LIN {X 0.170,Y -404.553,Z 1346.396,A 0.000,B 0.000,C 90.000,E1 287.221} C_DIS
LIN {X -0.116,Y -404.761,Z 1346.394,A 0.000,B 0.000,C 90.000,E1 286.913} C_DIS
LIN {X -0.219,Y -406.031,Z 1346.365,A 0.000,B 0.000,C 90.000,E1 281.715} C_DIS
LIN {X -0.210,Y -406.144,Z 1346.363,A 0.000,B 0.000,C 90.000,E1 281.366} C_DIS
LIN {X -0.106,Y -405.652,Z 1346.334,A 0.000,B 0.000,C 90.000,E1 276.144} C_DIS
LIN {X -0.101,Y -405.611,Z 1346.332,A 0.000,B 0.000,C 90.000,E1 275.796} C_DIS
LIN {X -0.028,Y -403.552,Z 1346.305,A 0.000,B 0.000,C 90.000,E1 270.917} C_DIS
LIN {X -0.092,Y -403.056,Z 1346.301,A 0.000,B 0.000,C 90.000,E1 270.229} C_DIS
LIN {X 0.132,Y -399.017,Z 1346.272,A 0.000,B 0.000,C 90.000,E1 264.951} C_DIS
LIN {X 0.026,Y -397.651,Z 1346.266,A 0.000,B 0.000,C 90.000,E1 263.913} C_DIS
LIN {X -0.094,Y -392.933,Z 1346.241,A 0.000,B 0.000,C 90.000,E1 259.342} C_DIS
LIN {X -0.136,Y -392.480,Z 1346.239,A 0.000,B 0.000,C 90.000,E1 258.993} C_DIS
LIN {X 0.013,Y -386.123,Z 1346.213,A 0.000,B 0.000,C 90.000,E1 254.338} C_DIS
LIN {X -0.028,Y -384.992,Z 1346.207,A 0.000,B 0.000,C 90.000,E1 253.268} C_DIS
LIN {X -0.154,Y -378.133,Z 1346.183,A 0.000,B 0.000,C 90.000,E1 248.954} C_DIS
LIN {X -0.065,Y -376.372,Z 1346.175,A 0.000,B 0.000,C 90.000,E1 247.486} C_DIS
LIN {X 0.060,Y -375.883,Z 1346.173,A 0.000,B 0.000,C 90.000,E1 247.102} C_DIS
LIN {X 0.010,Y -369.104,Z 1346.151,A 0.000,B 0.000,C 90.000,E1 243.076} C_DIS
LIN {X 0.089,Y -366.257,Z 1346.138,A 0.000,B 0.000,C 90.000,E1 240.845} C_DIS
LIN {X 0.050,Y -358.852,Z 1346.113,A 0.000,B 0.000,C 90.000,E1 236.373} C_DIS
LIN {X 0.038,Y -356.042,Z 1346.101,A 0.000,B 0.000,C 90.000,E1 234.116} C_DIS
LIN {X 0.034,Y -348.479,Z 1346.073,A 0.000,B 0.000,C 90.000,E1 229.175} C_DIS
LIN {X 0.095,Y -345.898,Z 1346.061,A 0.000,B 0.000,C 90.000,E1 226.863} C_DIS
LIN {X 0.062,Y -339.123,Z 1346.033,A 0.000,B 0.000,C 90.000,E1 221.838} C_DIS
LIN {X 0.145,Y -336.957,Z 1346.020,A 0.000,B 0.000,C 90.000,E1 219.483} C_DIS
LIN {X -0.034,Y -334.079,Z 1346.007,A 0.000,B 0.000,C 90.000,E1 217.202} C_DIS
LIN {X -0.051,Y -334.075,Z 1346.007,A 0.000,B 0.000,C 90.000,E1 217.202} C_DIS
LIN {X 0.031,Y -350.965,Z 1345.996,A 0.000,B 0.000,C 90.000,E1 215.185} C_DIS
LIN {X -0.024,Y -369.522,Z 1345.985,A 0.000,B 0.000,C 90.000,E1 213.245} C_DIS
LIN {X 0.079,Y -388.468,Z 1345.975,A 0.000,B 0.000,C 90.000,E1 211.465} C_DIS
LIN {X 0.012,Y -409.375,Z 1345.965,A 0.000,B 0.000,C 90.000,E1 209.745} C_DIS
LIN {X -0.255,Y -432.257,Z 1345.956,A 0.000,B 0.000,C 90.000,E1 208.103} C_DIS
LIN {X 0.054,Y -445.485,Z 1345.951,A 0.000,B 0.000,C 90.000,E1 207.180} C_DIS
LIN {X -0.207,Y -447.707,Z 1345.950,A 0.000,B 0.000,C 90.000,E1 207.001} C_DIS
LIN {X -0.015,Y -449.218,Z 1345.948,A 0.000,B 0.000,C 90.000,E1 206.693} C_DIS
LIN {X 0.051,Y -450.444,Z 1345.947,A 0.000,B 0.000,C 90.000,E1 206.360} C_DIS
LIN {X -0.075,Y -451.427,Z 1345.945,A 0.000,B 0.000,C 90.000,E1 206.052} C_DIS
LIN {X -0.118,Y -453.031,Z 1345.941,A 0.000,B 0.000,C 90.000,E1 205.412} C_DIS
LIN {X -0.151,Y -454.100,Z 1345.938,A 0.000,B 0.000,C 90.000,E1 204.771} C_DIS
LIN {X 0.033,Y -455.778,Z 1345.930,A 0.000,B 0.000,C 90.000,E1 203.462} C_DIS
LIN {X 0.063,Y -458.055,Z 1345.920,A 0.000,B 0.000,C 90.000,E1 201.535} C_DIS
LIN {X -0.205,Y -459.177,Z 1345.914,A 0.000,B 0.000,C 90.000,E1 200.610} C_DIS
LIN {X -0.077,Y -461.720,Z 1345.902,A 0.000,B 0.000,C 90.000,E1 198.362} C_DIS
LIN {X -0.023,Y -462.750,Z 1345.897,A 0.000,B 0.000,C 90.000,E1 197.402} C_DIS
LIN {X 0.202,Y -464.303,Z 1345.888,A 0.000,B 0.000,C 90.000,E1 195.788} C_DIS
LIN {X 0.054,Y -466.380,Z 1345.876,A 0.000,B 0.000,C 90.000,E1 193.592} C_DIS
LIN {X -0.076,Y -468.219,Z 1345.865,A 0.000,B 0.000,C 90.000,E1 191.715} C_DIS
LIN {X -0.254,Y -470.044,Z 1345.855,A 0.000,B 0.000,C 90.000,E1 189.849} C_DIS
LIN {X 0.135,Y -470.925,Z 1345.849,A 0.000,B 0.000,C 90.000,E1 188.859} C_DIS
LIN {X 0.107,Y -472.206,Z 1345.841,A 0.000,B 0.000,C 90.000,E1 187.296} C_DIS
LIN {X -0.248,Y -473.043,Z 1345.834,A 0.000,B 0.000,C 90.000,E1 186.087} C_DIS
LIN {X 0.107,Y -473.449,Z 1345.828,A 0.000,B 0.000,C 90.000,E1 185.106} C_DIS
LIN {X 0.241,Y -473.891,Z 1345.822,A 0.000,B 0.000,C 90.000,E1 183.841} C_DIS
LIN {X -0.126,Y -474.134,Z 1345.815,A 0.000,B 0.000,C 90.000,E1 182.636} C_DIS
LIN {X -0.016,Y -474.024,Z 1345.808,A 0.000,B 0.000,C 90.000,E1 181.375} C_DIS
LIN {X -0.181,Y -473.720,Z 1345.802,A 0.000,B 0.000,C 90.000,E1 180.458} C_DIS
LIN {X 0.126,Y -473.146,Z 1345.797,A 0.000,B 0.000,C 90.000,E1 179.484} C_DIS
LIN {X 0.206,Y -472.087,Z 1345.790,A 0.000,B 0.000,C 90.000,E1 178.224} C_DIS
LIN {X -0.192,Y -470.752,Z 1345.783,A 0.000,B 0.000,C 90.000,E1 177.020} C_DIS
LIN {X 0.091,Y -469.526,Z 1345.778,A 0.000,B 0.000,C 90.000,E1 176.045} C_DIS
LIN {X -0.071,Y -467.856,Z 1345.773,A 0.000,B 0.000,C 90.000,E1 175.122} C_DIS
LIN {X -0.043,Y -466.543,Z 1345.769,A 0.000,B 0.000,C 90.000,E1 174.489} C_DIS
LIN {X -0.026,Y -464.954,Z 1345.766,A 0.000,B 0.000,C 90.000,E1 173.856} C_DIS
LIN {X 0.182,Y -464.058,Z 1345.764,A 0.000,B 0.000,C 90.000,E1 173.514} C_DIS
LIN {X -0.036,Y -460.479,Z 1345.759,A 0.000,B 0.000,C 90.000,E1 172.591} C_DIS
LIN {X -0.010,Y -457.660,Z 1345.755,A 0.000,B 0.000,C 90.000,E1 171.951} C_DIS
LIN {X 0.143,Y -452.767,Z 1345.750,A 0.000,B 0.000,C 90.000,E1 170.971} C_DIS
LIN {X 0.244,Y -448.171,Z 1345.745,A 0.000,B 0.000,C 90.000,E1 170.151} C_DIS
LIN {X -0.083,Y -441.753,Z 1345.740,A 0.000,B 0.000,C 90.000,E1 169.218} C_DIS
LIN {X -0.218,Y -430.582,Z 1345.731,A 0.000,B 0.000,C 90.000,E1 167.589} C_DIS
LIN {X -0.058,Y -420.777,Z 1345.723,A 0.000,B 0.000,C 90.000,E1 166.061} C_DIS
LIN {X -0.011,Y -413.262,Z 1345.716,A 0.000,B 0.000,C 90.000,E1 164.866} C_DIS
LIN {X -0.056,Y -409.100,Z 1345.711,A 0.000,B 0.000,C 90.000,E1 164.031} C_DIS
LIN {X 0.156,Y -407.795,Z 1345.707,A 0.000,B 0.000,C 90.000,E1 163.268} C_DIS
LIN {X 0.118,Y -407.794,Z 1345.707,A 0.000,B 0.000,C 90.000,E1 163.268} C_DIS
LIN {X -0.092,Y -408.375,Z 1345.706,A 0.000,B 0.000,C 90.000,E1 163.087} C_DIS
LIN {X -0.078,Y -411.298,Z 1345.704,A 0.000,B 0.000,C 90.000,E1 162.653} C_DIS
LIN {X 0.071,Y -415.884,Z 1345.701,A 0.000,B 0.000,C 90.000,E1 162.127} C_DIS
LIN {X -0.127,Y -422.793,Z 1345.697,A 0.000,B 0.000,C 90.000,E1 161.511} C_DIS
LIN {X -0.205,Y -446.107,Z 1345.687,A 0.000,B 0.000,C 90.000,E1 159.699} C_DIS
LIN {X -0.083,Y -457.186,Z 1345.682,A 0.000,B 0.000,C 90.000,E1 158.847} C_DIS
LIN {X 0.010,Y -464.943,Z 1345.679,A 0.000,B 0.000,C 90.000,E1 158.230} C_DIS
LIN {X 0.070,Y -473.995,Z 1345.675,A 0.000,B 0.000,C 90.000,E1 157.486} C_DIS
LIN {X 0.028,Y -481.379,Z 1345.672,A 0.000,B 0.000,C 90.000,E1 156.869} C_DIS
LIN {X 0.099,Y -488.371,Z 1345.668,A 0.000,B 0.000,C 90.000,E1 156.230} C_DIS
LIN {X -0.060,Y -493.954,Z 1345.665,A 0.000,B 0.000,C 90.000,E1 155.717} C_DIS
LIN {X 0.040,Y -499.316,Z 1345.662,A 0.000,B 0.000,C 90.000,E1 155.177} C_DIS
LIN {X 0.115,Y -504.686,Z 1345.659,A 0.000,B 0.000,C 90.000,E1 154.613} C_DIS
LIN {X 0.140,Y -511.236,Z 1345.655,A 0.000,B 0.000,C 90.000,E1 153.896} C_DIS
LIN {X -0.009,Y -517.453,Z 1345.651,A 0.000,B 0.000,C 90.000,E1 153.179} C_DIS
LIN {X -0.220,Y -521.911,Z 1345.648,A 0.000,B 0.000,C 90.000,E1 152.615} C_DIS
LIN {X -0.159,Y -525.998,Z 1345.645,A 0.000,B 0.000,C 90.000,E1 152.025} C_DIS
LIN {X -0.067,Y -529.614,Z 1345.641,A 0.000,B 0.000,C 90.000,E1 151.435} C_DIS
LIN {X -0.093,Y -533.283,Z 1345.637,A 0.000,B 0.000,C 90.000,E1 150.717} C_DIS
LIN {X 0.056,Y -535.734,Z 1345.634,A 0.000,B 0.000,C 90.000,E1 150.127} C_DIS
LIN {X 0.220,Y -537.845,Z 1345.631,A 0.000,B 0.000,C 90.000,E1 149.537} C_DIS
LIN {X -0.343,Y -540.583,Z 1345.626,A 0.000,B 0.000,C 90.000,E1 148.742} C_DIS
LIN {X 0.135,Y -542.263,Z 1345.623,A 0.000,B 0.000,C 90.000,E1 148.122} C_DIS
LIN {X -0.095,Y -544.312,Z 1345.618,A 0.000,B 0.000,C 90.000,E1 147.296} C_DIS
LIN {X 0.155,Y -546.038,Z 1345.614,A 0.000,B 0.000,C 90.000,E1 146.421} C_DIS
LIN {X -0.035,Y -547.498,Z 1345.609,A 0.000,B 0.000,C 90.000,E1 145.595} C_DIS
LIN {X 0.054,Y -548.334,Z 1345.606,A 0.000,B 0.000,C 90.000,E1 145.022} C_DIS
LIN {X -0.062,Y -549.657,Z 1345.599,A 0.000,B 0.000,C 90.000,E1 143.909} C_DIS
LIN {X 0.162,Y -550.705,Z 1345.593,A 0.000,B 0.000,C 90.000,E1 142.763} C_DIS
LIN {X -0.035,Y -551.461,Z 1345.587,A 0.000,B 0.000,C 90.000,E1 141.662} C_DIS
LIN {X 0.379,Y -552.907,Z 1345.575,A 0.000,B 0.000,C 90.000,E1 139.380} C_DIS
LIN {X -0.141,Y -553.900,Z 1345.565,A 0.000,B 0.000,C 90.000,E1 137.757} C_DIS
LIN {X -0.205,Y -555.288,Z 1345.554,A 0.000,B 0.000,C 90.000,E1 135.810} C_DIS
LIN {X -0.220,Y -555.835,Z 1345.552,A 0.000,B 0.000,C 90.000,E1 135.324} C_DIS
LIN {X 0.002,Y -556.345,Z 1345.551,A 0.000,B 0.000,C 90.000,E1 135.162} C_DIS
LIN {X -0.102,Y -557.120,Z 1345.549,A 0.000,B 0.000,C 90.000,E1 134.838} C_DIS
LIN {X -0.144,Y -557.146,Z 1345.549,A 0.000,B 0.000,C 90.000,E1 134.838} C_DIS
LIN {X 0.106,Y -558.859,Z 1345.548,A 0.000,B 0.000,C 90.000,E1 134.595} C_DIS
LIN {X 0.291,Y -560.046,Z 1345.547,A 0.000,B 0.000,C 90.000,E1 134.514} C_DIS
LIN {X -0.276,Y -563.592,Z 1345.547,A 0.000,B 0.000,C 90.000,E1 134.433} C_DIS
LIN {X -0.342,Y -570.141,Z 1345.546,A 0.000,B 0.000,C 90.000,E1 134.271} C_DIS
LIN {X 0.031,Y -576.254,Z 1345.545,A 0.000,B 0.000,C 90.000,E1 134.028} C_DIS
LIN {X -0.356,Y -579.013,Z 1345.544,A 0.000,B 0.000,C 90.000,E1 133.947} C_DIS
LIN {X -0.199,Y -581.849,Z 1345.543,A 0.000,B 0.000,C 90.000,E1 133.785} C_DIS
LIN {X -0.033,Y -587.833,Z 1345.541,A 0.000,B 0.000,C 90.000,E1 133.419} C_DIS
LIN {X 0.071,Y -593.487,Z 1345.539,A 0.000,B 0.000,C 90.000,E1 133.014} C_DIS
LIN {X 0.242,Y -600.274,Z 1345.536,A 0.000,B 0.000,C 90.000,E1 132.447} C_DIS
LIN {X 0.007,Y -604.275,Z 1345.534,A 0.000,B 0.000,C 90.000,E1 132.123} C_DIS
LIN {X 0.042,Y -608.133,Z 1345.532,A 0.000,B 0.000,C 90.000,E1 131.757} C_DIS
LIN {X -0.044,Y -614.106,Z 1345.529,A 0.000,B 0.000,C 90.000,E1 131.148} C_DIS
LIN {X -0.248,Y -617.693,Z 1345.526,A 0.000,B 0.000,C 90.000,E1 130.782} C_DIS
LIN {X -0.047,Y -621.112,Z 1345.524,A 0.000,B 0.000,C 90.000,E1 130.378} C_DIS
LIN {X -0.085,Y -629.579,Z 1345.519,A 0.000,B 0.000,C 90.000,E1 129.358} C_DIS
LIN {X 0.281,Y -633.561,Z 1345.516,A 0.000,B 0.000,C 90.000,E1 128.830} C_DIS
LIN {X 0.010,Y -640.999,Z 1345.510,A 0.000,B 0.000,C 90.000,E1 127.855} C_DIS
LIN {X -0.169,Y -647.317,Z 1345.505,A 0.000,B 0.000,C 90.000,E1 126.996} C_DIS
LIN {X -0.109,Y -654.109,Z 1345.500,A 0.000,B 0.000,C 90.000,E1 126.011} C_DIS
LIN {X 0.081,Y -659.401,Z 1345.495,A 0.000,B 0.000,C 90.000,E1 125.152} C_DIS
LIN {X -0.317,Y -661.520,Z 1345.493,A 0.000,B 0.000,C 90.000,E1 124.818} C_DIS
LIN {X -0.274,Y -664.233,Z 1345.491,A 0.000,B 0.000,C 90.000,E1 124.326} C_DIS
LIN {X -0.152,Y -667.222,Z 1345.487,A 0.000,B 0.000,C 90.000,E1 123.706} C_DIS
LIN {X -0.078,Y -669.440,Z 1345.484,A 0.000,B 0.000,C 90.000,E1 123.214} C_DIS
LIN {X 0.158,Y -672.291,Z 1345.480,A 0.000,B 0.000,C 90.000,E1 122.467} C_DIS
LIN {X 0.067,Y -674.753,Z 1345.476,A 0.000,B 0.000,C 90.000,E1 121.750} C_DIS
LIN {X -0.042,Y -677.575,Z 1345.471,A 0.000,B 0.000,C 90.000,E1 120.797} C_DIS
LIN {X -0.069,Y -679.277,Z 1345.467,A 0.000,B 0.000,C 90.000,E1 120.079} C_DIS
LIN {X 0.259,Y -680.584,Z 1345.463,A 0.000,B 0.000,C 90.000,E1 119.333} C_DIS
LIN {X 0.061,Y -681.180,Z 1345.460,A 0.000,B 0.000,C 90.000,E1 118.871} C_DIS
LIN {X -0.134,Y -681.586,Z 1345.458,A 0.000,B 0.000,C 90.000,E1 118.409} C_DIS
LIN {X -0.125,Y -681.905,Z 1345.454,A 0.000,B 0.000,C 90.000,E1 117.692} C_DIS
LIN {X 0.183,Y -681.926,Z 1345.450,A 0.000,B 0.000,C 90.000,E1 116.950} C_DIS
LIN {X -0.208,Y -681.638,Z 1345.445,A 0.000,B 0.000,C 90.000,E1 116.027} C_DIS
LIN {X 0.113,Y -681.090,Z 1345.441,A 0.000,B 0.000,C 90.000,E1 115.283} C_DIS
LIN {X -0.097,Y -680.508,Z 1345.438,A 0.000,B 0.000,C 90.000,E1 114.823} C_DIS
LIN {X 0.022,Y -679.537,Z 1345.435,A 0.000,B 0.000,C 90.000,E1 114.335} C_DIS
LIN {X 0.415,Y -677.762,Z 1345.433,A 0.000,B 0.000,C 90.000,E1 113.823} C_DIS
LIN {X -0.286,Y -676.651,Z 1345.431,A 0.000,B 0.000,C 90.000,E1 113.643} C_DIS
LIN {X 0.184,Y -673.160,Z 1345.429,A 0.000,B 0.000,C 90.000,E1 113.153} C_DIS
LIN {X -0.346,Y -672.106,Z 1345.428,A 0.000,B 0.000,C 90.000,E1 113.078} C_DIS
LIN {X -0.258,Y -670.472,Z 1345.427,A 0.000,B 0.000,C 90.000,E1 112.950} C_DIS
LIN {X 0.297,Y -663.898,Z 1345.425,A 0.000,B 0.000,C 90.000,E1 112.514} C_DIS
LIN {X -0.134,Y -661.646,Z 1345.425,A 0.000,B 0.000,C 90.000,E1 112.461} C_DIS
LIN {X 0.299,Y -658.561,Z 1345.424,A 0.000,B 0.000,C 90.000,E1 112.333} C_DIS
LIN {X 0.252,Y -650.352,Z 1345.423,A 0.000,B 0.000,C 90.000,E1 112.153} C_DIS
LIN {X -0.169,Y -638.300,Z 1345.422,A 0.000,B 0.000,C 90.000,E1 111.950} C_DIS
LIN {X 0.373,Y -638.087,Z 1345.422,A 0.000,B 0.000,C 90.000,E1 111.897} C_DIS
LIN {X -0.028,Y -644.468,Z 1345.418,A 0.000,B 0.000,C 90.000,E1 111.153} C_DIS
LIN {X -0.166,Y -647.479,Z 1345.416,A 0.000,B 0.000,C 90.000,E1 110.791} C_DIS
LIN {X -0.291,Y -650.339,Z 1345.413,A 0.000,B 0.000,C 90.000,E1 110.429} C_DIS
LIN {X 0.343,Y -654.989,Z 1345.409,A 0.000,B 0.000,C 90.000,E1 109.631} C_DIS
LIN {X 0.261,Y -657.007,Z 1345.407,A 0.000,B 0.000,C 90.000,E1 109.268} C_DIS
LIN {X 0.074,Y -660.098,Z 1345.404,A 0.000,B 0.000,C 90.000,E1 108.671} C_DIS
LIN {X -0.034,Y -663.306,Z 1345.400,A 0.000,B 0.000,C 90.000,E1 107.946} C_DIS
LIN {X -0.115,Y -666.150,Z 1345.396,A 0.000,B 0.000,C 90.000,E1 107.221} C_DIS
LIN {X -0.092,Y -667.945,Z 1345.393,A 0.000,B 0.000,C 90.000,E1 106.732} C_DIS
LIN {X -0.325,Y -670.274,Z 1345.389,A 0.000,B 0.000,C 90.000,E1 106.024} C_DIS
LIN {X 0.297,Y -672.261,Z 1345.385,A 0.000,B 0.000,C 90.000,E1 105.245} C_DIS
LIN {X 0.171,Y -673.414,Z 1345.382,A 0.000,B 0.000,C 90.000,E1 104.773} C_DIS
LIN {X 0.055,Y -674.387,Z 1345.380,A 0.000,B 0.000,C 90.000,E1 104.300} C_DIS
LIN {X -0.056,Y -675.122,Z 1345.377,A 0.000,B 0.000,C 90.000,E1 103.828} C_DIS
LIN {X -0.213,Y -675.835,Z 1345.373,A 0.000,B 0.000,C 90.000,E1 103.119} C_DIS
LIN {X 0.344,Y -676.119,Z 1345.370,A 0.000,B 0.000,C 90.000,E1 102.591} C_DIS
LIN {X 0.190,Y -676.057,Z 1345.366,A 0.000,B 0.000,C 90.000,E1 101.883} C_DIS
LIN {X -0.049,Y -675.823,Z 1345.364,A 0.000,B 0.000,C 90.000,E1 101.422} C_DIS
LIN {X -0.155,Y -675.409,Z 1345.361,A 0.000,B 0.000,C 90.000,E1 100.950} C_DIS
LIN {X 0.215,Y -674.383,Z 1345.357,A 0.000,B 0.000,C 90.000,E1 100.197} C_DIS
LIN {X 0.093,Y -673.450,Z 1345.354,A 0.000,B 0.000,C 90.000,E1 99.726} C_DIS
LIN {X -0.150,Y -672.183,Z 1345.351,A 0.000,B 0.000,C 90.000,E1 99.265} C_DIS
LIN {X 0.268,Y -670.619,Z 1345.349,A 0.000,B 0.000,C 90.000,E1 98.746} C_DIS
LIN {X -0.067,Y -667.753,Z 1345.345,A 0.000,B 0.000,C 90.000,E1 98.049} C_DIS
LIN {X -0.336,Y -665.651,Z 1345.342,A 0.000,B 0.000,C 90.000,E1 97.587} C_DIS
LIN {X -0.250,Y -660.899,Z 1345.337,A 0.000,B 0.000,C 90.000,E1 96.606} C_DIS
LIN {X 0.065,Y -657.577,Z 1345.333,A 0.000,B 0.000,C 90.000,E1 95.967} C_DIS
LIN {X 0.276,Y -653.939,Z 1345.330,A 0.000,B 0.000,C 90.000,E1 95.334} C_DIS
LIN {X -0.194,Y -649.991,Z 1345.326,A 0.000,B 0.000,C 90.000,E1 94.759} C_DIS
LIN {X 0.017,Y -646.610,Z 1345.324,A 0.000,B 0.000,C 90.000,E1 94.245} C_DIS
LIN {X 0.252,Y -642.997,Z 1345.321,A 0.000,B 0.000,C 90.000,E1 93.726} C_DIS
LIN {X -0.099,Y -640.138,Z 1345.319,A 0.000,B 0.000,C 90.000,E1 93.383} C_DIS
LIN {X 0.087,Y -635.664,Z 1345.316,A 0.000,B 0.000,C 90.000,E1 92.865} C_DIS
LIN {X 0.129,Y -628.210,Z 1345.312,A 0.000,B 0.000,C 90.000,E1 92.121} C_DIS
LIN {X 0.071,Y -618.191,Z 1345.306,A 0.000,B 0.000,C 90.000,E1 91.146} C_DIS
LIN {X -0.199,Y -609.919,Z 1345.302,A 0.000,B 0.000,C 90.000,E1 90.458} C_DIS
LIN {X 0.135,Y -603.434,Z 1345.300,A 0.000,B 0.000,C 90.000,E1 90.000} C_DIS
LIN {X -0.295,Y -601.838,Z 1345.300,A 0.000,B 0.000,C 90.000,E1 89.943} C_DIS
LIN {X 0.275,Y -594.943,Z 1345.298,A 0.000,B 0.000,C 90.000,E1 89.542} C_DIS
LIN {X -0.130,Y -582.827,Z 1345.295,A 0.000,B 0.000,C 90.000,E1 89.083} C_DIS
LIN {X 0.231,Y -578.591,Z 1345.294,A 0.000,B 0.000,C 90.000,E1 88.854} C_DIS
LIN {X 0.040,Y -577.148,Z 1345.293,A 0.000,B 0.000,C 90.000,E1 88.797} C_DIS
LIN {X 0.144,Y -574.377,Z 1345.292,A 0.000,B 0.000,C 90.000,E1 88.568} C_DIS
LIN {X 0.073,Y -573.210,Z 1345.292,A 0.000,B 0.000,C 90.000,E1 88.453} C_DIS
LIN {X 0.037,Y -573.198,Z 1345.292,A 0.000,B 0.000,C 90.000,E1 88.453} C_DIS
LIN {X -0.140,Y -572.684,Z 1345.290,A 0.000,B 0.000,C 90.000,E1 88.224} C_DIS
LIN {X -0.238,Y -572.667,Z 1345.288,A 0.000,B 0.000,C 90.000,E1 87.936} C_DIS
LIN {X 0.117,Y -575.111,Z 1345.273,A 0.000,B 0.000,C 90.000,E1 85.179} C_DIS
LIN {X 0.112,Y -577.243,Z 1345.263,A 0.000,B 0.000,C 90.000,E1 83.280} C_DIS
LIN {X 0.082,Y -579.179,Z 1345.254,A 0.000,B 0.000,C 90.000,E1 81.659} C_DIS
LIN {X -0.136,Y -580.822,Z 1345.246,A 0.000,B 0.000,C 90.000,E1 80.330} C_DIS
LIN {X -0.242,Y -582.313,Z 1345.239,A 0.000,B 0.000,C 90.000,E1 78.993} C_DIS
LIN {X -0.210,Y -583.609,Z 1345.231,A 0.000,B 0.000,C 90.000,E1 77.645} C_DIS
LIN {X -0.018,Y -584.801,Z 1345.224,A 0.000,B 0.000,C 90.000,E1 76.284} C_DIS
LIN {X 0.052,Y -585.862,Z 1345.216,A 0.000,B 0.000,C 90.000,E1 74.936} C_DIS
LIN {X -0.122,Y -586.774,Z 1345.209,A 0.000,B 0.000,C 90.000,E1 73.614} C_DIS
LIN {X 0.293,Y -587.627,Z 1345.202,A 0.000,B 0.000,C 90.000,E1 72.236} C_DIS
LIN {X 0.126,Y -588.955,Z 1345.190,A 0.000,B 0.000,C 90.000,E1 70.115} C_DIS
LIN {X 0.188,Y -590.245,Z 1345.178,A 0.000,B 0.000,C 90.000,E1 67.975} C_DIS
LIN {X 0.289,Y -591.565,Z 1345.167,A 0.000,B 0.000,C 90.000,E1 66.102} C_DIS
LIN {X -0.025,Y -592.779,Z 1345.159,A 0.000,B 0.000,C 90.000,E1 64.537} C_DIS
LIN {X -0.071,Y -593.860,Z 1345.150,A 0.000,B 0.000,C 90.000,E1 62.948} C_DIS
LIN {X 0.273,Y -595.608,Z 1345.138,A 0.000,B 0.000,C 90.000,E1 60.795} C_DIS
LIN {X 0.204,Y -596.627,Z 1345.132,A 0.000,B 0.000,C 90.000,E1 59.744} C_DIS
LIN {X -0.149,Y -597.965,Z 1345.125,A 0.000,B 0.000,C 90.000,E1 58.456} C_DIS
LIN {X 0.267,Y -599.525,Z 1345.116,A 0.000,B 0.000,C 90.000,E1 56.834} C_DIS
LIN {X 0.203,Y -601.072,Z 1345.107,A 0.000,B 0.000,C 90.000,E1 55.261} C_DIS
LIN {X 0.355,Y -602.112,Z 1345.101,A 0.000,B 0.000,C 90.000,E1 54.196} C_DIS
LIN {X 0.190,Y -603.611,Z 1345.093,A 0.000,B 0.000,C 90.000,E1 52.637} C_DIS
LIN {X -0.103,Y -604.373,Z 1345.087,A 0.000,B 0.000,C 90.000,E1 51.618} C_DIS
LIN {X -0.006,Y -605.105,Z 1345.081,A 0.000,B 0.000,C 90.000,E1 50.561} C_DIS
LIN {X -0.024,Y -605.847,Z 1345.074,A 0.000,B 0.000,C 90.000,E1 49.256} C_DIS
LIN {X -0.361,Y -606.237,Z 1345.068,A 0.000,B 0.000,C 90.000,E1 48.243} C_DIS
LIN {X 0.169,Y -606.460,Z 1345.062,A 0.000,B 0.000,C 90.000,E1 47.148} C_DIS
LIN {X -0.345,Y -606.629,Z 1345.055,A 0.000,B 0.000,C 90.000,E1 45.891} C_DIS
LIN {X -0.245,Y -606.649,Z 1345.049,A 0.000,B 0.000,C 90.000,E1 44.838} C_DIS
LIN {X 0.044,Y -606.510,Z 1345.045,A 0.000,B 0.000,C 90.000,E1 44.028} C_DIS
LIN {X -0.088,Y -606.249,Z 1345.040,A 0.000,B 0.000,C 90.000,E1 43.257} C_DIS
LIN {X 0.055,Y -605.599,Z 1345.032,A 0.000,B 0.000,C 90.000,E1 41.676} C_DIS
LIN {X 0.226,Y -604.799,Z 1345.023,A 0.000,B 0.000,C 90.000,E1 40.092} C_DIS
LIN {X -0.218,Y -603.879,Z 1345.013,A 0.000,B 0.000,C 90.000,E1 38.302} C_DIS
LIN {X -0.033,Y -602.978,Z 1345.007,A 0.000,B 0.000,C 90.000,E1 37.237} C_DIS
LIN {X 0.147,Y -601.864,Z 1345.001,A 0.000,B 0.000,C 90.000,E1 36.171} C_DIS
LIN {X -0.283,Y -599.742,Z 1344.994,A 0.000,B 0.000,C 90.000,E1 34.898} C_DIS
LIN {X -0.259,Y -597.137,Z 1344.986,A 0.000,B 0.000,C 90.000,E1 33.579} C_DIS
LIN {X 0.095,Y -595.378,Z 1344.982,A 0.000,B 0.000,C 90.000,E1 32.752} C_DIS
LIN {X -0.183,Y -592.658,Z 1344.976,A 0.000,B 0.000,C 90.000,E1 31.720} C_DIS
LIN {X -0.115,Y -588.302,Z 1344.969,A 0.000,B 0.000,C 90.000,E1 30.384} C_DIS
LIN {X -0.344,Y -586.451,Z 1344.966,A 0.000,B 0.000,C 90.000,E1 29.873} C_DIS
LIN {X 0.250,Y -581.956,Z 1344.960,A 0.000,B 0.000,C 90.000,E1 28.743} C_DIS
LIN {X -0.081,Y -578.877,Z 1344.956,A 0.000,B 0.000,C 90.000,E1 28.103} C_DIS
LIN {X 0.190,Y -573.990,Z 1344.951,A 0.000,B 0.000,C 90.000,E1 27.129} C_DIS
LIN {X -0.288,Y -569.433,Z 1344.946,A 0.000,B 0.000,C 90.000,E1 26.360} C_DIS
LIN {X -0.119,Y -566.081,Z 1344.943,A 0.000,B 0.000,C 90.000,E1 25.796} C_DIS
LIN {X 0.170,Y -561.534,Z 1344.939,A 0.000,B 0.000,C 90.000,E1 25.079} C_DIS
LIN {X -0.126,Y -558.693,Z 1344.937,A 0.000,B 0.000,C 90.000,E1 24.695} C_DIS
LIN {X -0.146,Y -553.605,Z 1344.933,A 0.000,B 0.000,C 90.000,E1 24.003} C_DIS
LIN {X 0.294,Y -548.261,Z 1344.929,A 0.000,B 0.000,C 90.000,E1 23.259} C_DIS
LIN {X -0.032,Y -542.470,Z 1344.926,A 0.000,B 0.000,C 90.000,E1 22.589} C_DIS
LIN {X 0.318,Y -534.171,Z 1344.920,A 0.000,B 0.000,C 90.000,E1 21.589} C_DIS
LIN {X 0.142,Y -523.721,Z 1344.914,A 0.000,B 0.000,C 90.000,E1 20.482} C_DIS
LIN {X -0.160,Y -513.067,Z 1344.908,A 0.000,B 0.000,C 90.000,E1 19.396} C_DIS
LIN {X -0.153,Y -503.917,Z 1344.902,A 0.000,B 0.000,C 90.000,E1 18.417} C_DIS
LIN {X 0.171,Y -493.056,Z 1344.896,A 0.000,B 0.000,C 90.000,E1 17.275} C_DIS
LIN {X -0.125,Y -482.889,Z 1344.891,A 0.000,B 0.000,C 90.000,E1 16.370} C_DIS
LIN {X -0.081,Y -473.040,Z 1344.886,A 0.000,B 0.000,C 90.000,E1 15.426} C_DIS
LIN {X 0.037,Y -461.483,Z 1344.880,A 0.000,B 0.000,C 90.000,E1 14.300} C_DIS
LIN {X 0.122,Y -444.300,Z 1344.870,A 0.000,B 0.000,C 90.000,E1 12.591} C_DIS
LIN {X 0.083,Y -421.676,Z 1344.857,A 0.000,B 0.000,C 90.000,E1 10.197} C_DIS
LIN {X -0.035,Y -406.105,Z 1344.847,A 0.000,B 0.000,C 90.000,E1 8.454} C_DIS
LIN {X 0.091,Y -399.224,Z 1344.843,A 0.000,B 0.000,C 90.000,E1 7.644} C_DIS
LIN {X -0.124,Y -396.614,Z 1344.841,A 0.000,B 0.000,C 90.000,E1 7.352} C_DIS
LIN {X -0.020,Y -394.822,Z 1344.839,A 0.000,B 0.000,C 90.000,E1 7.004} C_DIS
LIN {X 0.067,Y -394.611,Z 1344.839,A 0.000,B 0.000,C 90.000,E1 6.947} C_DIS
LIN {X 0.029,Y -394.640,Z 1344.839,A 0.000,B 0.000,C 90.000,E1 6.947} C_DIS
LIN {X -0.061,Y -395.617,Z 1344.838,A 0.000,B 0.000,C 90.000,E1 6.834} C_DIS
LIN {X 0.177,Y -399.215,Z 1344.836,A 0.000,B 0.000,C 90.000,E1 6.486} C_DIS
LIN {X -0.131,Y -407.101,Z 1344.833,A 0.000,B 0.000,C 90.000,E1 5.967} C_DIS
LIN {X -0.083,Y -410.469,Z 1344.832,A 0.000,B 0.000,C 90.000,E1 5.739} C_DIS
LIN {X 0.005,Y -416.857,Z 1344.829,A 0.000,B 0.000,C 90.000,E1 5.277} C_DIS
LIN {X -0.181,Y -422.858,Z 1344.827,A 0.000,B 0.000,C 90.000,E1 4.816} C_DIS
LIN {X 0.144,Y -429.901,Z 1344.823,A 0.000,B 0.000,C 90.000,E1 4.131} C_DIS
LIN {X -0.170,Y -437.080,Z 1344.819,A 0.000,B 0.000,C 90.000,E1 3.440} C_DIS
LIN {X -0.144,Y -445.349,Z 1344.814,A 0.000,B 0.000,C 90.000,E1 2.522} C_DIS
LIN {X -0.224,Y -449.390,Z 1344.811,A 0.000,B 0.000,C 90.000,E1 2.064} C_DIS
LIN {X -0.202,Y -455.542,Z 1344.807,A 0.000,B 0.000,C 90.000,E1 1.318} C_DIS
LIN {X 0.068,Y -459.323,Z 1344.805,A 0.000,B 0.000,C 90.000,E1 0.802} C_DIS
LIN {X 0.005,Y -464.115,Z 1344.801,A 0.000,B 0.000,C 90.000,E1 0.172} C_DIS
LIN {X 0.052,Y -470.027,Z 1344.796,A 0.000,B 0.000,C 90.000,E1 359.312} C_DIS
LIN {X 0.196,Y -475.051,Z 1344.792,A 0.000,B 0.000,C 90.000,E1 358.511} C_DIS
LIN {X -0.072,Y -479.691,Z 1344.788,A 0.000,B 0.000,C 90.000,E1 357.764} C_DIS
LIN {X 0.163,Y -484.023,Z 1344.783,A 0.000,B 0.000,C 90.000,E1 356.963} C_DIS
LIN {X -0.176,Y -487.302,Z 1344.780,A 0.000,B 0.000,C 90.000,E1 356.388} C_DIS
LIN {X 0.161,Y -490.974,Z 1344.776,A 0.000,B 0.000,C 90.000,E1 355.584} C_DIS
LIN {X 0.042,Y -494.324,Z 1344.771,A 0.000,B 0.000,C 90.000,E1 354.837} C_DIS
LIN {X 0.177,Y -498.135,Z 1344.766,A 0.000,B 0.000,C 90.000,E1 353.913} C_DIS
LIN {X -0.057,Y -500.453,Z 1344.763,A 0.000,B 0.000,C 90.000,E1 353.337} C_DIS
LIN {X 0.218,Y -502.631,Z 1344.760,A 0.000,B 0.000,C 90.000,E1 352.704} C_DIS
LIN {X 0.007,Y -504.643,Z 1344.756,A 0.000,B 0.000,C 90.000,E1 352.129} C_DIS
LIN {X -0.176,Y -507.348,Z 1344.751,A 0.000,B 0.000,C 90.000,E1 351.254} C_DIS
LIN {X 0.098,Y -509.729,Z 1344.746,A 0.000,B 0.000,C 90.000,E1 350.330} C_DIS
LIN {X -0.053,Y -512.593,Z 1344.740,A 0.000,B 0.000,C 90.000,E1 349.162} C_DIS
LIN {X -0.160,Y -515.062,Z 1344.733,A 0.000,B 0.000,C 90.000,E1 347.993} C_DIS
LIN {X -0.202,Y -516.196,Z 1344.730,A 0.000,B 0.000,C 90.000,E1 347.409} C_DIS
LIN {X -0.146,Y -518.073,Z 1344.723,A 0.000,B 0.000,C 90.000,E1 346.228} C_DIS
LIN {X -0.050,Y -519.285,Z 1344.719,A 0.000,B 0.000,C 90.000,E1 345.338} C_DIS
LIN {X 0.059,Y -520.215,Z 1344.714,A 0.000,B 0.000,C 90.000,E1 344.448} C_DIS
LIN {X 0.041,Y -520.752,Z 1344.710,A 0.000,B 0.000,C 90.000,E1 343.866} C_DIS
LIN {X -0.200,Y -521.393,Z 1344.704,A 0.000,B 0.000,C 90.000,E1 342.725} C_DIS
LIN {X 0.063,Y -521.579,Z 1344.698,A 0.000,B 0.000,C 90.000,E1 341.529} C_DIS
LIN {X -0.132,Y -521.515,Z 1344.694,A 0.000,B 0.000,C 90.000,E1 340.967} C_DIS
LIN {X 0.150,Y -521.112,Z 1344.689,A 0.000,B 0.000,C 90.000,E1 340.061} C_DIS
LIN {X -0.217,Y -520.692,Z 1344.686,A 0.000,B 0.000,C 90.000,E1 339.518} C_DIS
LIN {X 0.232,Y -519.704,Z 1344.681,A 0.000,B 0.000,C 90.000,E1 338.592} C_DIS
LIN {X 0.190,Y -518.300,Z 1344.676,A 0.000,B 0.000,C 90.000,E1 337.720} C_DIS
LIN {X 0.134,Y -517.750,Z 1344.675,A 0.000,B 0.000,C 90.000,E1 337.433} C_DIS
LIN {X -0.203,Y -517.069,Z 1344.673,A 0.000,B 0.000,C 90.000,E1 337.177} C_DIS
LIN {X -0.066,Y -516.202,Z 1344.672,A 0.000,B 0.000,C 90.000,E1 336.869} C_DIS
LIN {X 0.067,Y -515.141,Z 1344.670,A 0.000,B 0.000,C 90.000,E1 336.561} C_DIS
LIN {X -0.068,Y -513.708,Z 1344.668,A 0.000,B 0.000,C 90.000,E1 336.282} C_DIS
LIN {X 0.230,Y -512.701,Z 1344.667,A 0.000,B 0.000,C 90.000,E1 336.102} C_DIS
LIN {X 0.058,Y -511.284,Z 1344.667,A 0.000,B 0.000,C 90.000,E1 335.973} C_DIS
LIN {X 0.110,Y -500.873,Z 1344.664,A 0.000,B 0.000,C 90.000,E1 335.433} C_DIS
LIN {X 0.114,Y -472.825,Z 1344.655,A 0.000,B 0.000,C 90.000,E1 333.896} C_DIS
LIN {X 0.095,Y -446.789,Z 1344.646,A 0.000,B 0.000,C 90.000,E1 332.281} C_DIS
LIN {X 0.100,Y -422.753,Z 1344.637,A 0.000,B 0.000,C 90.000,E1 330.589} C_DIS
LIN {X -0.148,Y -400.714,Z 1344.627,A 0.000,B 0.000,C 90.000,E1 328.869} C_DIS
LIN {X 0.016,Y -380.645,Z 1344.617,A 0.000,B 0.000,C 90.000,E1 327.041} C_DIS
LIN {X -0.162,Y -369.913,Z 1344.611,A 0.000,B 0.000,C 90.000,E1 326.008} C_DIS
LIN {X 0.114,Y -369.900,Z 1344.611,A 0.000,B 0.000,C 90.000,E1 325.960} C_DIS
LIN {X 0.054,Y -371.678,Z 1344.602,A 0.000,B 0.000,C 90.000,E1 324.356} C_DIS
LIN {X -0.182,Y -377.238,Z 1344.568,A 0.000,B 0.000,C 90.000,E1 318.162} C_DIS
LIN {X 0.096,Y -378.170,Z 1344.563,A 0.000,B 0.000,C 90.000,E1 317.391} C_DIS
LIN {X 0.083,Y -383.815,Z 1344.531,A 0.000,B 0.000,C 90.000,E1 311.595} C_DIS
LIN {X -0.123,Y -384.806,Z 1344.527,A 0.000,B 0.000,C 90.000,E1 310.906} C_DIS
LIN {X -0.134,Y -390.975,Z 1344.493,A 0.000,B 0.000,C 90.000,E1 304.818} C_DIS
LIN {X -0.067,Y -391.375,Z 1344.491,A 0.000,B 0.000,C 90.000,E1 304.452} C_DIS
LIN {X 0.202,Y -396.706,Z 1344.460,A 0.000,B 0.000,C 90.000,E1 298.743} C_DIS
LIN {X -0.119,Y -397.081,Z 1344.458,A 0.000,B 0.000,C 90.000,E1 298.437} C_DIS
LIN {X -0.163,Y -401.504,Z 1344.427,A 0.000,B 0.000,C 90.000,E1 292.823} C_DIS
LIN {X 0.154,Y -401.772,Z 1344.423,A 0.000,B 0.000,C 90.000,E1 292.078} C_DIS
LIN {X -0.037,Y -404.579,Z 1344.396,A 0.000,B 0.000,C 90.000,E1 287.221} C_DIS
LIN {X 0.064,Y -404.759,Z 1344.394,A 0.000,B 0.000,C 90.000,E1 286.858} C_DIS
LIN {X -0.029,Y -406.048,Z 1344.365,A 0.000,B 0.000,C 90.000,E1 281.658} C_DIS
LIN {X 0.060,Y -406.131,Z 1344.363,A 0.000,B 0.000,C 90.000,E1 281.299} C_DIS
LIN {X 0.090,Y -405.659,Z 1344.334,A 0.000,B 0.000,C 90.000,E1 276.087} C_DIS
LIN {X 0.096,Y -405.591,Z 1344.332,A 0.000,B 0.000,C 90.000,E1 275.739} C_DIS
LIN {X 0.169,Y -403.545,Z 1344.305,A 0.000,B 0.000,C 90.000,E1 270.859} C_DIS
LIN {X 0.104,Y -403.024,Z 1344.301,A 0.000,B 0.000,C 90.000,E1 270.172} C_DIS
LIN {X -0.074,Y -399.003,Z 1344.272,A 0.000,B 0.000,C 90.000,E1 264.951} C_DIS
LIN {X 0.088,Y -392.912,Z 1344.241,A 0.000,B 0.000,C 90.000,E1 259.285} C_DIS
LIN {X 0.078,Y -391.844,Z 1344.237,A 0.000,B 0.000,C 90.000,E1 258.578} C_DIS
LIN {X -0.167,Y -385.716,Z 1344.211,A 0.000,B 0.000,C 90.000,E1 253.976} C_DIS
LIN {X -0.120,Y -384.939,Z 1344.207,A 0.000,B 0.000,C 90.000,E1 253.251} C_DIS
LIN {X -0.003,Y -378.093,Z 1344.183,A 0.000,B 0.000,C 90.000,E1 248.901} C_DIS
LIN {X 0.081,Y -376.338,Z 1344.175,A 0.000,B 0.000,C 90.000,E1 247.433} C_DIS
LIN {X -0.141,Y -375.822,Z 1344.173,A 0.000,B 0.000,C 90.000,E1 247.102} C_DIS
LIN {X -0.023,Y -369.061,Z 1344.150,A 0.000,B 0.000,C 90.000,E1 243.050} C_DIS
LIN {X -0.111,Y -366.212,Z 1344.138,A 0.000,B 0.000,C 90.000,E1 240.845} C_DIS
LIN {X 0.051,Y -358.808,Z 1344.113,A 0.000,B 0.000,C 90.000,E1 236.342} C_DIS
LIN {X 0.129,Y -355.999,Z 1344.101,A 0.000,B 0.000,C 90.000,E1 234.069} C_DIS
LIN {X -0.065,Y -348.920,Z 1344.075,A 0.000,B 0.000,C 90.000,E1 229.542} C_DIS
LIN {X -0.100,Y -345.845,Z 1344.060,A 0.000,B 0.000,C 90.000,E1 226.863} C_DIS
LIN {X -0.132,Y -339.088,Z 1344.032,A 0.000,B 0.000,C 90.000,E1 221.838} C_DIS
LIN {X -0.049,Y -336.931,Z 1344.019,A 0.000,B 0.000,C 90.000,E1 219.483} C_DIS
LIN {X -0.014,Y -335.520,Z 1344.013,A 0.000,B 0.000,C 90.000,E1 218.382} C_DIS
LIN {X -0.031,Y -335.540,Z 1344.013,A 0.000,B 0.000,C 90.000,E1 218.382} C_DIS
LIN {X -0.037,Y -352.480,Z 1344.002,A 0.000,B 0.000,C 90.000,E1 216.297} C_DIS
LIN {X 0.119,Y -370.795,Z 1343.991,A 0.000,B 0.000,C 90.000,E1 214.278} C_DIS
LIN {X 0.144,Y -389.519,Z 1343.981,A 0.000,B 0.000,C 90.000,E1 212.467} C_DIS
LIN {X -0.044,Y -410.208,Z 1343.971,A 0.000,B 0.000,C 90.000,E1 210.718} C_DIS
LIN {X -0.084,Y -432.877,Z 1343.961,A 0.000,B 0.000,C 90.000,E1 208.999} C_DIS
LIN {X -0.176,Y -445.958,Z 1343.956,A 0.000,B 0.000,C 90.000,E1 208.103} C_DIS
LIN {X 0.080,Y -447.732,Z 1343.955,A 0.000,B 0.000,C 90.000,E1 207.847} C_DIS
LIN {X 0.142,Y -449.290,Z 1343.953,A 0.000,B 0.000,C 90.000,E1 207.513} C_DIS
LIN {X 0.008,Y -450.428,Z 1343.951,A 0.000,B 0.000,C 90.000,E1 207.206} C_DIS
LIN {X 0.082,Y -451.338,Z 1343.949,A 0.000,B 0.000,C 90.000,E1 206.873} C_DIS
LIN {X 0.037,Y -452.728,Z 1343.946,A 0.000,B 0.000,C 90.000,E1 206.232} C_DIS
LIN {X -0.108,Y -454.331,Z 1343.940,A 0.000,B 0.000,C 90.000,E1 205.283} C_DIS
LIN {X 0.168,Y -456.417,Z 1343.932,A 0.000,B 0.000,C 90.000,E1 203.643} C_DIS
LIN {X -0.126,Y -458.350,Z 1343.923,A 0.000,B 0.000,C 90.000,E1 202.078} C_DIS
LIN {X -0.050,Y -459.929,Z 1343.916,A 0.000,B 0.000,C 90.000,E1 200.791} C_DIS
LIN {X -0.183,Y -461.709,Z 1343.907,A 0.000,B 0.000,C 90.000,E1 199.214} C_DIS
LIN {X -0.203,Y -463.220,Z 1343.900,A 0.000,B 0.000,C 90.000,E1 197.946} C_DIS
LIN {X -0.205,Y -464.628,Z 1343.893,A 0.000,B 0.000,C 90.000,E1 196.677} C_DIS
LIN {X 0.024,Y -467.043,Z 1343.879,A 0.000,B 0.000,C 90.000,E1 194.120} C_DIS
LIN {X 0.183,Y -469.220,Z 1343.866,A 0.000,B 0.000,C 90.000,E1 191.895} C_DIS
LIN {X 0.117,Y -471.116,Z 1343.856,A 0.000,B 0.000,C 90.000,E1 190.018} C_DIS
LIN {X -0.199,Y -472.310,Z 1343.849,A 0.000,B 0.000,C 90.000,E1 188.803} C_DIS
LIN {X -0.199,Y -473.668,Z 1343.840,A 0.000,B 0.000,C 90.000,E1 187.239} C_DIS
LIN {X -0.010,Y -474.530,Z 1343.833,A 0.000,B 0.000,C 90.000,E1 185.967} C_DIS
LIN {X -0.080,Y -475.252,Z 1343.825,A 0.000,B 0.000,C 90.000,E1 184.416} C_DIS
LIN {X -0.134,Y -475.704,Z 1343.816,A 0.000,B 0.000,C 90.000,E1 182.865} C_DIS
LIN {X -0.001,Y -475.688,Z 1343.809,A 0.000,B 0.000,C 90.000,E1 181.604} C_DIS
LIN {X -0.148,Y -475.488,Z 1343.804,A 0.000,B 0.000,C 90.000,E1 180.688} C_DIS
LIN {X 0.180,Y -475.074,Z 1343.799,A 0.000,B 0.000,C 90.000,E1 179.714} C_DIS
LIN {X 0.093,Y -473.894,Z 1343.790,A 0.000,B 0.000,C 90.000,E1 178.165} C_DIS
LIN {X 0.178,Y -472.598,Z 1343.783,A 0.000,B 0.000,C 90.000,E1 176.906} C_DIS
LIN {X 0.011,Y -471.466,Z 1343.778,A 0.000,B 0.000,C 90.000,E1 175.988} C_DIS
LIN {X -0.130,Y -470.032,Z 1343.773,A 0.000,B 0.000,C 90.000,E1 175.065} C_DIS
LIN {X -0.086,Y -468.779,Z 1343.769,A 0.000,B 0.000,C 90.000,E1 174.432} C_DIS
LIN {X 0.165,Y -466.374,Z 1343.764,A 0.000,B 0.000,C 90.000,E1 173.457} C_DIS
LIN {X 0.233,Y -464.416,Z 1343.760,A 0.000,B 0.000,C 90.000,E1 172.818} C_DIS
LIN {X 0.104,Y -459.785,Z 1343.754,A 0.000,B 0.000,C 90.000,E1 171.724} C_DIS
LIN {X -0.247,Y -455.812,Z 1343.750,A 0.000,B 0.000,C 90.000,E1 170.971} C_DIS
LIN {X -0.112,Y -451.321,Z 1343.745,A 0.000,B 0.000,C 90.000,E1 170.151} C_DIS
LIN {X -0.152,Y -447.280,Z 1343.742,A 0.000,B 0.000,C 90.000,E1 169.511} C_DIS
LIN {X -0.177,Y -441.891,Z 1343.737,A 0.000,B 0.000,C 90.000,E1 168.701} C_DIS
LIN {X -0.118,Y -429.735,Z 1343.727,A 0.000,B 0.000,C 90.000,E1 166.881} C_DIS
LIN {X -0.047,Y -422.159,Z 1343.721,A 0.000,B 0.000,C 90.000,E1 165.700} C_DIS
LIN {X 0.192,Y -417.764,Z 1343.717,A 0.000,B 0.000,C 90.000,E1 164.991} C_DIS
LIN {X 0.051,Y -413.897,Z 1343.713,A 0.000,B 0.000,C 90.000,E1 164.338} C_DIS
LIN {X 0.195,Y -412.338,Z 1343.711,A 0.000,B 0.000,C 90.000,E1 163.976} C_DIS
LIN {X -0.117,Y -410.702,Z 1343.709,A 0.000,B 0.000,C 90.000,E1 163.559} C_DIS
LIN {X -0.049,Y -410.308,Z 1343.708,A 0.000,B 0.000,C 90.000,E1 163.378} C_DIS
LIN {X 0.071,Y -410.504,Z 1343.705,A 0.000,B 0.000,C 90.000,E1 162.960} C_DIS
LIN {X 0.043,Y -410.524,Z 1343.705,A 0.000,B 0.000,C 90.000,E1 162.960} C_DIS
LIN {X -0.009,Y -411.805,Z 1343.704,A 0.000,B 0.000,C 90.000,E1 162.725} C_DIS
LIN {X -0.099,Y -412.623,Z 1343.703,A 0.000,B 0.000,C 90.000,E1 162.543} C_DIS
LIN {X 0.191,Y -415.478,Z 1343.701,A 0.000,B 0.000,C 90.000,E1 162.181} C_DIS
LIN {X -0.060,Y -416.730,Z 1343.700,A 0.000,B 0.000,C 90.000,E1 162.054} C_DIS
LIN {X -0.107,Y -423.216,Z 1343.697,A 0.000,B 0.000,C 90.000,E1 161.456} C_DIS
LIN {X -0.028,Y -435.232,Z 1343.692,A 0.000,B 0.000,C 90.000,E1 160.477} C_DIS
LIN {X -0.071,Y -447.945,Z 1343.686,A 0.000,B 0.000,C 90.000,E1 159.518} C_DIS
LIN {X 0.072,Y -458.960,Z 1343.682,A 0.000,B 0.000,C 90.000,E1 158.666} C_DIS
LIN {X -0.208,Y -464.997,Z 1343.679,A 0.000,B 0.000,C 90.000,E1 158.230} C_DIS
LIN {X -0.192,Y -475.694,Z 1343.674,A 0.000,B 0.000,C 90.000,E1 157.358} C_DIS
LIN {X 0.286,Y -483.074,Z 1343.671,A 0.000,B 0.000,C 90.000,E1 156.666} C_DIS
LIN {X 0.013,Y -488.852,Z 1343.668,A 0.000,B 0.000,C 90.000,E1 156.177} C_DIS
LIN {X 0.086,Y -497.309,Z 1343.663,A 0.000,B 0.000,C 90.000,E1 155.357} C_DIS
LIN {X 0.082,Y -504.073,Z 1343.659,A 0.000,B 0.000,C 90.000,E1 154.665} C_DIS
LIN {X 0.087,Y -510.669,Z 1343.655,A 0.000,B 0.000,C 90.000,E1 153.948} C_DIS
LIN {X 0.105,Y -514.441,Z 1343.653,A 0.000,B 0.000,C 90.000,E1 153.512} C_DIS
LIN {X 0.046,Y -518.065,Z 1343.651,A 0.000,B 0.000,C 90.000,E1 153.076} C_DIS
LIN {X 0.076,Y -522.458,Z 1343.647,A 0.000,B 0.000,C 90.000,E1 152.487} C_DIS
LIN {X 0.300,Y -525.580,Z 1343.645,A 0.000,B 0.000,C 90.000,E1 152.025} C_DIS
LIN {X 0.242,Y -530.055,Z 1343.641,A 0.000,B 0.000,C 90.000,E1 151.307} C_DIS
LIN {X 0.109,Y -532.958,Z 1343.638,A 0.000,B 0.000,C 90.000,E1 150.745} C_DIS
LIN {X -0.091,Y -536.005,Z 1343.634,A 0.000,B 0.000,C 90.000,E1 150.049} C_DIS
LIN {X 0.077,Y -538.052,Z 1343.630,A 0.000,B 0.000,C 90.000,E1 149.459} C_DIS
LIN {X -0.022,Y -540.699,Z 1343.626,A 0.000,B 0.000,C 90.000,E1 148.614} C_DIS
LIN {X -0.003,Y -542.329,Z 1343.623,A 0.000,B 0.000,C 90.000,E1 148.043} C_DIS
LIN {X 0.228,Y -544.327,Z 1343.618,A 0.000,B 0.000,C 90.000,E1 147.168} C_DIS
LIN {X 0.022,Y -546.034,Z 1343.613,A 0.000,B 0.000,C 90.000,E1 146.342} C_DIS
LIN {X -0.167,Y -547.475,Z 1343.608,A 0.000,B 0.000,C 90.000,E1 145.515} C_DIS
LIN {X 0.374,Y -548.266,Z 1343.605,A 0.000,B 0.000,C 90.000,E1 144.895} C_DIS
LIN {X -0.191,Y -549.574,Z 1343.599,A 0.000,B 0.000,C 90.000,E1 143.829} C_DIS
LIN {X 0.034,Y -550.550,Z 1343.593,A 0.000,B 0.000,C 90.000,E1 142.683} C_DIS
LIN {X -0.103,Y -551.462,Z 1343.585,A 0.000,B 0.000,C 90.000,E1 141.295} C_DIS
LIN {X -0.170,Y -552.562,Z 1343.576,A 0.000,B 0.000,C 90.000,E1 139.622} C_DIS
LIN {X 0.078,Y -553.565,Z 1343.566,A 0.000,B 0.000,C 90.000,E1 137.919} C_DIS
LIN {X 0.006,Y -555.099,Z 1343.555,A 0.000,B 0.000,C 90.000,E1 135.972} C_DIS
LIN {X -0.026,Y -555.478,Z 1343.555,A 0.000,B 0.000,C 90.000,E1 135.810} C_DIS
LIN {X 0.018,Y -556.039,Z 1343.552,A 0.000,B 0.000,C 90.000,E1 135.405} C_DIS
LIN {X 0.070,Y -556.949,Z 1343.551,A 0.000,B 0.000,C 90.000,E1 135.243} C_DIS
LIN {X -0.258,Y -557.825,Z 1343.550,A 0.000,B 0.000,C 90.000,E1 135.081} C_DIS
LIN {X -0.300,Y -557.886,Z 1343.550,A 0.000,B 0.000,C 90.000,E1 135.081} C_DIS
LIN {X -0.274,Y -559.662,Z 1343.550,A 0.000,B 0.000,C 90.000,E1 135.000} C_DIS
LIN {X -0.320,Y -571.558,Z 1343.548,A 0.000,B 0.000,C 90.000,E1 134.676} C_DIS
LIN {X -0.082,Y -577.516,Z 1343.547,A 0.000,B 0.000,C 90.000,E1 134.433} C_DIS
LIN {X 0.008,Y -586.403,Z 1343.544,A 0.000,B 0.000,C 90.000,E1 133.947} C_DIS
LIN {X 0.310,Y -591.988,Z 1343.542,A 0.000,B 0.000,C 90.000,E1 133.542} C_DIS
LIN {X 0.070,Y -598.766,Z 1343.539,A 0.000,B 0.000,C 90.000,E1 133.014} C_DIS
LIN {X -0.148,Y -602.785,Z 1343.537,A 0.000,B 0.000,C 90.000,E1 132.690} C_DIS
LIN {X -0.102,Y -606.735,Z 1343.535,A 0.000,B 0.000,C 90.000,E1 132.324} C_DIS
LIN {X -0.177,Y -611.697,Z 1343.532,A 0.000,B 0.000,C 90.000,E1 131.838} C_DIS
LIN {X 0.328,Y -617.574,Z 1343.529,A 0.000,B 0.000,C 90.000,E1 131.148} C_DIS
LIN {X 0.002,Y -622.084,Z 1343.526,A 0.000,B 0.000,C 90.000,E1 130.663} C_DIS
LIN {X -0.028,Y -630.411,Z 1343.520,A 0.000,B 0.000,C 90.000,E1 129.644} C_DIS
LIN {X 0.190,Y -635.293,Z 1343.517,A 0.000,B 0.000,C 90.000,E1 128.991} C_DIS
LIN {X 0.350,Y -641.743,Z 1343.512,A 0.000,B 0.000,C 90.000,E1 128.096} C_DIS
LIN {X -0.129,Y -649.586,Z 1343.506,A 0.000,B 0.000,C 90.000,E1 127.030} C_DIS
LIN {X -0.207,Y -655.426,Z 1343.501,A 0.000,B 0.000,C 90.000,E1 126.171} C_DIS
LIN {X -0.173,Y -661.464,Z 1343.495,A 0.000,B 0.000,C 90.000,E1 125.185} C_DIS
LIN {X 0.367,Y -665.388,Z 1343.491,A 0.000,B 0.000,C 90.000,E1 124.405} C_DIS
LIN {X 0.436,Y -667.774,Z 1343.489,A 0.000,B 0.000,C 90.000,E1 123.913} C_DIS
LIN {X 0.099,Y -671.007,Z 1343.485,A 0.000,B 0.000,C 90.000,E1 123.214} C_DIS
LIN {X -0.011,Y -673.679,Z 1343.481,A 0.000,B 0.000,C 90.000,E1 122.498} C_DIS
LIN {X -0.301,Y -676.010,Z 1343.477,A 0.000,B 0.000,C 90.000,E1 121.799} C_DIS
LIN {X 0.182,Y -678.691,Z 1343.471,A 0.000,B 0.000,C 90.000,E1 120.797} C_DIS
LIN {X 0.167,Y -680.321,Z 1343.467,A 0.000,B 0.000,C 90.000,E1 120.079} C_DIS
LIN {X -0.422,Y -681.563,Z 1343.463,A 0.000,B 0.000,C 90.000,E1 119.411} C_DIS
LIN {X -0.016,Y -682.174,Z 1343.461,A 0.000,B 0.000,C 90.000,E1 118.899} C_DIS
LIN {X 0.009,Y -682.665,Z 1343.457,A 0.000,B 0.000,C 90.000,E1 118.180} C_DIS
LIN {X -0.174,Y -682.896,Z 1343.454,A 0.000,B 0.000,C 90.000,E1 117.719} C_DIS
LIN {X -0.148,Y -682.932,Z 1343.450,A 0.000,B 0.000,C 90.000,E1 117.001} C_DIS
LIN {X 0.083,Y -682.687,Z 1343.445,A 0.000,B 0.000,C 90.000,E1 116.027} C_DIS
LIN {X -0.202,Y -682.143,Z 1343.441,A 0.000,B 0.000,C 90.000,E1 115.335} C_DIS
LIN {X -0.076,Y -681.594,Z 1343.438,A 0.000,B 0.000,C 90.000,E1 114.847} C_DIS
LIN {X -0.284,Y -680.576,Z 1343.435,A 0.000,B 0.000,C 90.000,E1 114.387} C_DIS
LIN {X -0.083,Y -679.829,Z 1343.434,A 0.000,B 0.000,C 90.000,E1 114.131} C_DIS
LIN {X 0.036,Y -677.938,Z 1343.431,A 0.000,B 0.000,C 90.000,E1 113.643} C_DIS
LIN {X 0.132,Y -677.116,Z 1343.431,A 0.000,B 0.000,C 90.000,E1 113.515} C_DIS
LIN {X 0.146,Y -674.192,Z 1343.429,A 0.000,B 0.000,C 90.000,E1 113.153} C_DIS
LIN {X 0.046,Y -672.159,Z 1343.428,A 0.000,B 0.000,C 90.000,E1 112.950} C_DIS
LIN {X 0.132,Y -670.113,Z 1343.427,A 0.000,B 0.000,C 90.000,E1 112.823} C_DIS
LIN {X -0.041,Y -667.790,Z 1343.426,A 0.000,B 0.000,C 90.000,E1 112.717} C_DIS
LIN {X -0.285,Y -663.962,Z 1343.425,A 0.000,B 0.000,C 90.000,E1 112.514} C_DIS
LIN {X 0.031,Y -659.438,Z 1343.424,A 0.000,B 0.000,C 90.000,E1 112.333} C_DIS
LIN {X -0.152,Y -652.935,Z 1343.423,A 0.000,B 0.000,C 90.000,E1 112.206} C_DIS
LIN {X 0.256,Y -638.823,Z 1343.422,A 0.000,B 0.000,C 90.000,E1 111.897} C_DIS
LIN {X 0.207,Y -638.763,Z 1343.422,A 0.000,B 0.000,C 90.000,E1 111.897} C_DIS
LIN {X -0.199,Y -642.397,Z 1343.419,A 0.000,B 0.000,C 90.000,E1 111.461} C_DIS
LIN {X 0.282,Y -646.602,Z 1343.416,A 0.000,B 0.000,C 90.000,E1 110.918} C_DIS
LIN {X 0.194,Y -650.415,Z 1343.414,A 0.000,B 0.000,C 90.000,E1 110.429} C_DIS
LIN {X 0.041,Y -655.126,Z 1343.410,A 0.000,B 0.000,C 90.000,E1 109.704} C_DIS
LIN {X 0.008,Y -657.804,Z 1343.407,A 0.000,B 0.000,C 90.000,E1 109.214} C_DIS
LIN {X -0.009,Y -660.265,Z 1343.404,A 0.000,B 0.000,C 90.000,E1 108.725} C_DIS
LIN {X -0.119,Y -663.497,Z 1343.400,A 0.000,B 0.000,C 90.000,E1 108.000} C_DIS
LIN {X -0.201,Y -666.358,Z 1343.396,A 0.000,B 0.000,C 90.000,E1 107.275} C_DIS
LIN {X -0.372,Y -668.145,Z 1343.393,A 0.000,B 0.000,C 90.000,E1 106.804} C_DIS
LIN {X 0.232,Y -670.497,Z 1343.389,A 0.000,B 0.000,C 90.000,E1 106.024} C_DIS
LIN {X 0.031,Y -672.483,Z 1343.385,A 0.000,B 0.000,C 90.000,E1 105.315} C_DIS
LIN {X 0.083,Y -673.646,Z 1343.382,A 0.000,B 0.000,C 90.000,E1 104.828} C_DIS
LIN {X -0.033,Y -674.638,Z 1343.380,A 0.000,B 0.000,C 90.000,E1 104.356} C_DIS
LIN {X -0.197,Y -675.697,Z 1343.376,A 0.000,B 0.000,C 90.000,E1 103.647} C_DIS
LIN {X 0.357,Y -676.171,Z 1343.373,A 0.000,B 0.000,C 90.000,E1 103.119} C_DIS
LIN {X 0.258,Y -676.427,Z 1343.370,A 0.000,B 0.000,C 90.000,E1 102.647} C_DIS
LIN {X -0.035,Y -676.450,Z 1343.366,A 0.000,B 0.000,C 90.000,E1 101.951} C_DIS
LIN {X -0.134,Y -676.271,Z 1343.364,A 0.000,B 0.000,C 90.000,E1 101.478} C_DIS
LIN {X -0.239,Y -675.859,Z 1343.361,A 0.000,B 0.000,C 90.000,E1 101.007} C_DIS
LIN {X 0.191,Y -675.253,Z 1343.358,A 0.000,B 0.000,C 90.000,E1 100.489} C_DIS
LIN {X -0.099,Y -673.972,Z 1343.354,A 0.000,B 0.000,C 90.000,E1 99.792} C_DIS
LIN {X -0.225,Y -672.754,Z 1343.352,A 0.000,B 0.000,C 90.000,E1 99.321} C_DIS
LIN {X 0.195,Y -671.198,Z 1343.349,A 0.000,B 0.000,C 90.000,E1 98.803} C_DIS
LIN {X -0.134,Y -668.369,Z 1343.345,A 0.000,B 0.000,C 90.000,E1 98.106} C_DIS
LIN {X 0.260,Y -666.306,Z 1343.342,A 0.000,B 0.000,C 90.000,E1 97.587} C_DIS
LIN {X -0.306,Y -661.571,Z 1343.337,A 0.000,B 0.000,C 90.000,E1 96.663} C_DIS
LIN {X -0.055,Y -658.266,Z 1343.333,A 0.000,B 0.000,C 90.000,E1 96.030} C_DIS
LIN {X 0.230,Y -654.636,Z 1343.330,A 0.000,B 0.000,C 90.000,E1 95.391} C_DIS
LIN {X -0.184,Y -651.533,Z 1343.327,A 0.000,B 0.000,C 90.000,E1 94.935} C_DIS
LIN {X -0.020,Y -647.308,Z 1343.324,A 0.000,B 0.000,C 90.000,E1 94.302} C_DIS
LIN {X 0.219,Y -643.725,Z 1343.321,A 0.000,B 0.000,C 90.000,E1 93.784} C_DIS
LIN {X -0.128,Y -640.879,Z 1343.319,A 0.000,B 0.000,C 90.000,E1 93.440} C_DIS
LIN {X -0.062,Y -635.324,Z 1343.316,A 0.000,B 0.000,C 90.000,E1 92.808} C_DIS
LIN {X -0.006,Y -627.797,Z 1343.312,A 0.000,B 0.000,C 90.000,E1 92.064} C_DIS
LIN {X -0.050,Y -617.747,Z 1343.306,A 0.000,B 0.000,C 90.000,E1 91.088} C_DIS
LIN {X -0.273,Y -609.441,Z 1343.302,A 0.000,B 0.000,C 90.000,E1 90.401} C_DIS
LIN {X 0.219,Y -603.055,Z 1343.300,A 0.000,B 0.000,C 90.000,E1 89.943} C_DIS
LIN {X -0.270,Y -597.779,Z 1343.298,A 0.000,B 0.000,C 90.000,E1 89.714} C_DIS
LIN {X -0.192,Y -594.348,Z 1343.297,A 0.000,B 0.000,C 90.000,E1 89.542} C_DIS
LIN {X -0.143,Y -580.704,Z 1343.294,A 0.000,B 0.000,C 90.000,E1 88.969} C_DIS
LIN {X 0.243,Y -577.799,Z 1343.293,A 0.000,B 0.000,C 90.000,E1 88.797} C_DIS
LIN {X -0.147,Y -575.621,Z 1343.293,A 0.000,B 0.000,C 90.000,E1 88.682} C_DIS
LIN {X -0.256,Y -573.530,Z 1343.292,A 0.000,B 0.000,C 90.000,E1 88.511} C_DIS
LIN {X -0.052,Y -573.239,Z 1343.291,A 0.000,B 0.000,C 90.000,E1 88.453} C_DIS
LIN {X -0.089,Y -573.212,Z 1343.291,A 0.000,B 0.000,C 90.000,E1 88.453} C_DIS
LIN {X 0.066,Y -572.630,Z 1343.290,A 0.000,B 0.000,C 90.000,E1 88.165} C_DIS
LIN {X 0.262,Y -572.742,Z 1343.287,A 0.000,B 0.000,C 90.000,E1 87.593} C_DIS
LIN {X -0.283,Y -574.755,Z 1343.275,A 0.000,B 0.000,C 90.000,E1 85.469} C_DIS
LIN {X -0.105,Y -577.155,Z 1343.263,A 0.000,B 0.000,C 90.000,E1 83.280} C_DIS
LIN {X -0.138,Y -579.107,Z 1343.254,A 0.000,B 0.000,C 90.000,E1 81.659} C_DIS
LIN {X 0.085,Y -580.451,Z 1343.248,A 0.000,B 0.000,C 90.000,E1 80.557} C_DIS
LIN {X -0.015,Y -581.943,Z 1343.240,A 0.000,B 0.000,C 90.000,E1 79.218} C_DIS
LIN {X 0.233,Y -583.067,Z 1343.234,A 0.000,B 0.000,C 90.000,E1 78.117} C_DIS
LIN {X 0.082,Y -584.484,Z 1343.225,A 0.000,B 0.000,C 90.000,E1 76.520} C_DIS
LIN {X -0.090,Y -585.375,Z 1343.219,A 0.000,B 0.000,C 90.000,E1 75.463} C_DIS
LIN {X 0.133,Y -586.308,Z 1343.212,A 0.000,B 0.000,C 90.000,E1 74.102} C_DIS
LIN {X -0.029,Y -587.233,Z 1343.204,A 0.000,B 0.000,C 90.000,E1 72.779} C_DIS
LIN {X 0.154,Y -587.847,Z 1343.198,A 0.000,B 0.000,C 90.000,E1 71.692} C_DIS
LIN {X -0.109,Y -588.897,Z 1343.190,A 0.000,B 0.000,C 90.000,E1 70.115} C_DIS
LIN {X -0.049,Y -590.169,Z 1343.178,A 0.000,B 0.000,C 90.000,E1 67.975} C_DIS
LIN {X 0.049,Y -591.455,Z 1343.167,A 0.000,B 0.000,C 90.000,E1 66.102} C_DIS
LIN {X -0.267,Y -592.683,Z 1343.158,A 0.000,B 0.000,C 90.000,E1 64.537} C_DIS
LIN {X -0.045,Y -593.769,Z 1343.150,A 0.000,B 0.000,C 90.000,E1 62.922} C_DIS
LIN {X -0.068,Y -595.796,Z 1343.136,A 0.000,B 0.000,C 90.000,E1 60.539} C_DIS
LIN {X 0.045,Y -596.367,Z 1343.133,A 0.000,B 0.000,C 90.000,E1 59.999} C_DIS
LIN {X 0.334,Y -598.132,Z 1343.123,A 0.000,B 0.000,C 90.000,E1 58.122} C_DIS
LIN {X -0.081,Y -599.708,Z 1343.114,A 0.000,B 0.000,C 90.000,E1 56.580} C_DIS
LIN {X 0.193,Y -601.303,Z 1343.106,A 0.000,B 0.000,C 90.000,E1 54.975} C_DIS
LIN {X -0.240,Y -602.519,Z 1343.098,A 0.000,B 0.000,C 90.000,E1 53.703} C_DIS
LIN {X -0.068,Y -603.552,Z 1343.092,A 0.000,B 0.000,C 90.000,E1 52.637} C_DIS
LIN {X -0.363,Y -604.312,Z 1343.087,A 0.000,B 0.000,C 90.000,E1 51.618} C_DIS
LIN {X 0.201,Y -605.064,Z 1343.081,A 0.000,B 0.000,C 90.000,E1 50.517} C_DIS
LIN {X 0.110,Y -605.799,Z 1343.073,A 0.000,B 0.000,C 90.000,E1 49.218} C_DIS
LIN {X 0.232,Y -606.196,Z 1343.068,A 0.000,B 0.000,C 90.000,E1 48.162} C_DIS
LIN {X 0.098,Y -606.358,Z 1343.063,A 0.000,B 0.000,C 90.000,E1 47.391} C_DIS
LIN {X 0.248,Y -606.577,Z 1343.055,A 0.000,B 0.000,C 90.000,E1 45.810} C_DIS
LIN {X -0.083,Y -606.562,Z 1343.049,A 0.000,B 0.000,C 90.000,E1 44.798} C_DIS
LIN {X -0.221,Y -606.417,Z 1343.045,A 0.000,B 0.000,C 90.000,E1 44.028} C_DIS
LIN {X 0.061,Y -606.153,Z 1343.040,A 0.000,B 0.000,C 90.000,E1 43.218} C_DIS
LIN {X -0.213,Y -605.518,Z 1343.031,A 0.000,B 0.000,C 90.000,E1 41.676} C_DIS
LIN {X 0.159,Y -604.908,Z 1343.024,A 0.000,B 0.000,C 90.000,E1 40.334} C_DIS
LIN {X -0.015,Y -603.836,Z 1343.013,A 0.000,B 0.000,C 90.000,E1 38.257} C_DIS
LIN {X -0.304,Y -602.927,Z 1343.007,A 0.000,B 0.000,C 90.000,E1 37.237} C_DIS
LIN {X -0.124,Y -601.801,Z 1343.001,A 0.000,B 0.000,C 90.000,E1 36.171} C_DIS
LIN {X 0.281,Y -599.673,Z 1342.994,A 0.000,B 0.000,C 90.000,E1 34.818} C_DIS
LIN {X 0.297,Y -597.081,Z 1342.986,A 0.000,B 0.000,C 90.000,E1 33.499} C_DIS
LIN {X -0.175,Y -595.341,Z 1342.982,A 0.000,B 0.000,C 90.000,E1 32.752} C_DIS
LIN {X 0.052,Y -592.623,Z 1342.976,A 0.000,B 0.000,C 90.000,E1 31.671} C_DIS
LIN {X 0.123,Y -588.264,Z 1342.969,A 0.000,B 0.000,C 90.000,E1 30.335} C_DIS
LIN {X 0.188,Y -586.386,Z 1342.966,A 0.000,B 0.000,C 90.000,E1 29.795} C_DIS
LIN {X -0.017,Y -581.879,Z 1342.960,A 0.000,B 0.000,C 90.000,E1 28.743} C_DIS
LIN {X -0.347,Y -578.790,Z 1342.956,A 0.000,B 0.000,C 90.000,E1 28.103} C_DIS
LIN {X 0.000,Y -574.600,Z 1342.952,A 0.000,B 0.000,C 90.000,E1 27.257} C_DIS
LIN {X -0.309,Y -571.650,Z 1342.948,A 0.000,B 0.000,C 90.000,E1 26.744} C_DIS
LIN {X -0.041,Y -569.309,Z 1342.946,A 0.000,B 0.000,C 90.000,E1 26.309} C_DIS
LIN {X -0.137,Y -565.950,Z 1342.943,A 0.000,B 0.000,C 90.000,E1 25.771} C_DIS
LIN {X 0.004,Y -562.337,Z 1342.940,A 0.000,B 0.000,C 90.000,E1 25.207} C_DIS
LIN {X 0.120,Y -558.495,Z 1342.937,A 0.000,B 0.000,C 90.000,E1 24.643} C_DIS
LIN {X 0.209,Y -554.449,Z 1342.934,A 0.000,B 0.000,C 90.000,E1 24.079} C_DIS
LIN {X 0.151,Y -549.133,Z 1342.930,A 0.000,B 0.000,C 90.000,E1 23.387} C_DIS
LIN {X 0.170,Y -544.599,Z 1342.927,A 0.000,B 0.000,C 90.000,E1 22.823} C_DIS
LIN {X -0.206,Y -536.339,Z 1342.922,A 0.000,B 0.000,C 90.000,E1 21.897} C_DIS
LIN {X -0.133,Y -532.510,Z 1342.919,A 0.000,B 0.000,C 90.000,E1 21.461} C_DIS
LIN {X -0.150,Y -523.368,Z 1342.914,A 0.000,B 0.000,C 90.000,E1 20.482} C_DIS
LIN {X 0.142,Y -512.858,Z 1342.908,A 0.000,B 0.000,C 90.000,E1 19.341} C_DIS
LIN {X 0.159,Y -503.678,Z 1342.902,A 0.000,B 0.000,C 90.000,E1 18.362} C_DIS
LIN {X 0.186,Y -493.018,Z 1342.896,A 0.000,B 0.000,C 90.000,E1 17.275} C_DIS
LIN {X -0.170,Y -475.942,Z 1342.887,A 0.000,B 0.000,C 90.000,E1 15.717} C_DIS
LIN {X 0.126,Y -461.476,Z 1342.880,A 0.000,B 0.000,C 90.000,E1 14.300} C_DIS
LIN {X -0.046,Y -445.708,Z 1342.871,A 0.000,B 0.000,C 90.000,E1 12.771} C_DIS
LIN {X -0.107,Y -424.356,Z 1342.859,A 0.000,B 0.000,C 90.000,E1 10.546} C_DIS
LIN {X -0.169,Y -410.253,Z 1342.850,A 0.000,B 0.000,C 90.000,E1 8.973} C_DIS
LIN {X 0.179,Y -404.559,Z 1342.846,A 0.000,B 0.000,C 90.000,E1 8.276} C_DIS
LIN {X -0.023,Y -397.977,Z 1342.842,A 0.000,B 0.000,C 90.000,E1 7.530} C_DIS
LIN {X -0.169,Y -395.964,Z 1342.840,A 0.000,B 0.000,C 90.000,E1 7.296} C_DIS
LIN {X 0.073,Y -394.724,Z 1342.839,A 0.000,B 0.000,C 90.000,E1 7.004} C_DIS
LIN {X 0.035,Y -394.713,Z 1342.839,A 0.000,B 0.000,C 90.000,E1 7.004} C_DIS
LIN {X -0.002,Y -394.712,Z 1342.839,A 0.000,B 0.000,C 90.000,E1 7.004} C_DIS
LIN {X -0.041,Y -394.745,Z 1342.839,A 0.000,B 0.000,C 90.000,E1 7.004} C_DIS
LIN {X -0.181,Y -395.217,Z 1342.839,A 0.000,B 0.000,C 90.000,E1 6.947} C_DIS
LIN {X 0.117,Y -398.570,Z 1342.837,A 0.000,B 0.000,C 90.000,E1 6.606} C_DIS
LIN {X -0.049,Y -406.002,Z 1342.834,A 0.000,B 0.000,C 90.000,E1 6.087} C_DIS
LIN {X -0.163,Y -412.267,Z 1342.832,A 0.000,B 0.000,C 90.000,E1 5.682} C_DIS
LIN {X -0.167,Y -417.231,Z 1342.830,A 0.000,B 0.000,C 90.000,E1 5.334} C_DIS
LIN {X -0.025,Y -423.392,Z 1342.827,A 0.000,B 0.000,C 90.000,E1 4.821} C_DIS
LIN {X 0.190,Y -429.439,Z 1342.824,A 0.000,B 0.000,C 90.000,E1 4.245} C_DIS
LIN {X 0.105,Y -438.111,Z 1342.819,A 0.000,B 0.000,C 90.000,E1 3.383} C_DIS
LIN {X 0.034,Y -445.042,Z 1342.815,A 0.000,B 0.000,C 90.000,E1 2.636} C_DIS
LIN {X 0.136,Y -450.410,Z 1342.811,A 0.000,B 0.000,C 90.000,E1 2.007} C_DIS
LIN {X -0.032,Y -454.048,Z 1342.809,A 0.000,B 0.000,C 90.000,E1 1.604} C_DIS
LIN {X 0.003,Y -460.398,Z 1342.805,A 0.000,B 0.000,C 90.000,E1 0.802} C_DIS
LIN {X 0.000,Y -466.307,Z 1342.800,A 0.000,B 0.000,C 90.000,E1 360.000} C_DIS
LIN {X 0.058,Y -471.063,Z 1342.796,A 0.000,B 0.000,C 90.000,E1 359.312} C_DIS
LIN {X 0.212,Y -476.058,Z 1342.792,A 0.000,B 0.000,C 90.000,E1 358.511} C_DIS
LIN {X -0.046,Y -480.731,Z 1342.788,A 0.000,B 0.000,C 90.000,E1 357.764} C_DIS
LIN {X 0.200,Y -485.032,Z 1342.783,A 0.000,B 0.000,C 90.000,E1 356.963} C_DIS
LIN {X -0.132,Y -488.311,Z 1342.780,A 0.000,B 0.000,C 90.000,E1 356.388} C_DIS
LIN {X 0.215,Y -491.975,Z 1342.776,A 0.000,B 0.000,C 90.000,E1 355.584} C_DIS
LIN {X -0.001,Y -496.634,Z 1342.770,A 0.000,B 0.000,C 90.000,E1 354.546} C_DIS
LIN {X 0.109,Y -500.363,Z 1342.765,A 0.000,B 0.000,C 90.000,E1 353.628} C_DIS
LIN {X -0.191,Y -503.682,Z 1342.760,A 0.000,B 0.000,C 90.000,E1 352.761} C_DIS
LIN {X 0.044,Y -506.636,Z 1342.755,A 0.000,B 0.000,C 90.000,E1 351.837} C_DIS
LIN {X -0.065,Y -508.409,Z 1342.751,A 0.000,B 0.000,C 90.000,E1 351.254} C_DIS
LIN {X 0.223,Y -510.788,Z 1342.746,A 0.000,B 0.000,C 90.000,E1 350.330} C_DIS
LIN {X 0.088,Y -513.656,Z 1342.740,A 0.000,B 0.000,C 90.000,E1 349.162} C_DIS
LIN {X 0.038,Y -514.969,Z 1342.737,A 0.000,B 0.000,C 90.000,E1 348.578} C_DIS
LIN {X -0.035,Y -517.317,Z 1342.730,A 0.000,B 0.000,C 90.000,E1 347.409} C_DIS
LIN {X 0.037,Y -519.187,Z 1342.724,A 0.000,B 0.000,C 90.000,E1 346.228} C_DIS
LIN {X 0.014,Y -520.393,Z 1342.719,A 0.000,B 0.000,C 90.000,E1 345.353} C_DIS
LIN {X 0.128,Y -521.354,Z 1342.714,A 0.000,B 0.000,C 90.000,E1 344.464} C_DIS
LIN {X -0.101,Y -522.076,Z 1342.709,A 0.000,B 0.000,C 90.000,E1 343.614} C_DIS
LIN {X 0.033,Y -522.551,Z 1342.704,A 0.000,B 0.000,C 90.000,E1 342.725} C_DIS
LIN {X -0.182,Y -522.716,Z 1342.698,A 0.000,B 0.000,C 90.000,E1 341.583} C_DIS
LIN {X 0.128,Y -522.677,Z 1342.694,A 0.000,B 0.000,C 90.000,E1 340.967} C_DIS
LIN {X -0.092,Y -522.088,Z 1342.688,A 0.000,B 0.000,C 90.000,E1 339.826} C_DIS
LIN {X -0.114,Y -521.269,Z 1342.683,A 0.000,B 0.000,C 90.000,E1 338.954} C_DIS
LIN {X 0.151,Y -520.016,Z 1342.678,A 0.000,B 0.000,C 90.000,E1 338.050} C_DIS
LIN {X -0.225,Y -517.978,Z 1342.672,A 0.000,B 0.000,C 90.000,E1 336.922} C_DIS
LIN {X -0.085,Y -517.348,Z 1342.670,A 0.000,B 0.000,C 90.000,E1 336.613} C_DIS
LIN {X 0.053,Y -516.567,Z 1342.668,A 0.000,B 0.000,C 90.000,E1 336.305} C_DIS
LIN {X -0.284,Y -515.531,Z 1342.667,A 0.000,B 0.000,C 90.000,E1 336.049} C_DIS
LIN {X -0.323,Y -513.604,Z 1342.664,A 0.000,B 0.000,C 90.000,E1 335.613} C_DIS
LIN {X 0.186,Y -512.780,Z 1342.664,A 0.000,B 0.000,C 90.000,E1 335.409} C_DIS
LIN {X 0.013,Y -511.739,Z 1342.663,A 0.000,B 0.000,C 90.000,E1 335.281} C_DIS
LIN {X -0.159,Y -510.290,Z 1342.662,A 0.000,B 0.000,C 90.000,E1 335.153} C_DIS
LIN {X -0.003,Y -475.559,Z 1342.651,A 0.000,B 0.000,C 90.000,E1 333.204} C_DIS
LIN {X -0.047,Y -449.688,Z 1342.642,A 0.000,B 0.000,C 90.000,E1 331.563} C_DIS
LIN {X -0.254,Y -425.823,Z 1342.632,A 0.000,B 0.000,C 90.000,E1 329.871} C_DIS
LIN {X -0.132,Y -403.957,Z 1342.623,A 0.000,B 0.000,C 90.000,E1 328.074} C_DIS
LIN {X 0.069,Y -384.064,Z 1342.612,A 0.000,B 0.000,C 90.000,E1 326.215} C_DIS
LIN {X 0.032,Y -371.055,Z 1342.605,A 0.000,B 0.000,C 90.000,E1 324.895} C_DIS
LIN {X 0.000,Y -371.058,Z 1342.605,A 0.000,B 0.000,C 90.000,E1 324.895} C_DIS
LIN {X -0.021,Y -371.726,Z 1342.602,A 0.000,B 0.000,C 90.000,E1 324.322} C_DIS
LIN {X 0.059,Y -377.294,Z 1342.567,A 0.000,B 0.000,C 90.000,E1 318.081} C_DIS
LIN {X -0.196,Y -378.204,Z 1342.563,A 0.000,B 0.000,C 90.000,E1 317.391} C_DIS
LIN {X 0.075,Y -383.874,Z 1342.531,A 0.000,B 0.000,C 90.000,E1 311.553} C_DIS
LIN {X -0.126,Y -384.852,Z 1342.527,A 0.000,B 0.000,C 90.000,E1 310.862} C_DIS
LIN {X 0.047,Y -390.544,Z 1342.495,A 0.000,B 0.000,C 90.000,E1 305.105} C_DIS
LIN {X 0.114,Y -391.036,Z 1342.493,A 0.000,B 0.000,C 90.000,E1 304.739} C_DIS
LIN {X -0.040,Y -391.400,Z 1342.491,A 0.000,B 0.000,C 90.000,E1 304.405} C_DIS
LIN {X -0.096,Y -396.763,Z 1342.460,A 0.000,B 0.000,C 90.000,E1 298.743} C_DIS
LIN {X 0.122,Y -397.099,Z 1342.458,A 0.000,B 0.000,C 90.000,E1 298.359} C_DIS
LIN {X -0.092,Y -401.552,Z 1342.427,A 0.000,B 0.000,C 90.000,E1 292.770} C_DIS
LIN {X 0.050,Y -404.617,Z 1342.396,A 0.000,B 0.000,C 90.000,E1 287.166} C_DIS
LIN {X 0.152,Y -404.755,Z 1342.394,A 0.000,B 0.000,C 90.000,E1 286.804} C_DIS
LIN {X 0.150,Y -406.072,Z 1342.365,A 0.000,B 0.000,C 90.000,E1 281.591} C_DIS
LIN {X 0.159,Y -406.114,Z 1342.363,A 0.000,B 0.000,C 90.000,E1 281.243} C_DIS
LIN {X -0.209,Y -405.669,Z 1342.334,A 0.000,B 0.000,C 90.000,E1 276.087} C_DIS
LIN {X 0.199,Y -405.559,Z 1342.332,A 0.000,B 0.000,C 90.000,E1 275.682} C_DIS
LIN {X -0.130,Y -403.525,Z 1342.305,A 0.000,B 0.000,C 90.000,E1 270.859} C_DIS
LIN {X -0.163,Y -403.316,Z 1342.303,A 0.000,B 0.000,C 90.000,E1 270.516} C_DIS
LIN {X 0.026,Y -398.974,Z 1342.272,A 0.000,B 0.000,C 90.000,E1 264.894} C_DIS
LIN {X -0.168,Y -393.145,Z 1342.242,A 0.000,B 0.000,C 90.000,E1 259.634} C_DIS
LIN {X -0.135,Y -392.880,Z 1342.240,A 0.000,B 0.000,C 90.000,E1 259.275} C_DIS
LIN {X -0.113,Y -386.045,Z 1342.213,A 0.000,B 0.000,C 90.000,E1 254.283} C_DIS
LIN {X -0.067,Y -385.314,Z 1342.209,A 0.000,B 0.000,C 90.000,E1 253.559} C_DIS
LIN {X -0.045,Y -384.858,Z 1342.207,A 0.000,B 0.000,C 90.000,E1 253.196} C_DIS
LIN {X 0.057,Y -378.035,Z 1342.183,A 0.000,B 0.000,C 90.000,E1 248.847} C_DIS
LIN {X -0.066,Y -376.288,Z 1342.174,A 0.000,B 0.000,C 90.000,E1 247.411} C_DIS
LIN {X -0.087,Y -375.736,Z 1342.172,A 0.000,B 0.000,C 90.000,E1 247.050} C_DIS
LIN {X 0.017,Y -368.998,Z 1342.150,A 0.000,B 0.000,C 90.000,E1 242.999} C_DIS
LIN {X -0.080,Y -366.140,Z 1342.138,A 0.000,B 0.000,C 90.000,E1 240.795} C_DIS
LIN {X -0.174,Y -359.268,Z 1342.115,A 0.000,B 0.000,C 90.000,E1 236.707} C_DIS
LIN {X 0.052,Y -355.930,Z 1342.100,A 0.000,B 0.000,C 90.000,E1 234.036} C_DIS
LIN {X 0.143,Y -348.860,Z 1342.075,A 0.000,B 0.000,C 90.000,E1 229.461} C_DIS
LIN {X -0.017,Y -346.237,Z 1342.062,A 0.000,B 0.000,C 90.000,E1 227.187} C_DIS
LIN {X 0.106,Y -345.769,Z 1342.060,A 0.000,B 0.000,C 90.000,E1 226.782} C_DIS
LIN {X 0.066,Y -339.039,Z 1342.032,A 0.000,B 0.000,C 90.000,E1 221.757} C_DIS
LIN {X 0.041,Y -337.007,Z 1342.020,A 0.000,B 0.000,C 90.000,E1 219.564} C_DIS
LIN {X 0.023,Y -337.026,Z 1342.020,A 0.000,B 0.000,C 90.000,E1 219.564} C_DIS
LIN {X -0.080,Y -352.696,Z 1342.009,A 0.000,B 0.000,C 90.000,E1 217.569} C_DIS
LIN {X -0.102,Y -370.725,Z 1341.997,A 0.000,B 0.000,C 90.000,E1 215.518} C_DIS
LIN {X 0.067,Y -389.190,Z 1341.987,A 0.000,B 0.000,C 90.000,E1 213.627} C_DIS
LIN {X 0.033,Y -409.612,Z 1341.977,A 0.000,B 0.000,C 90.000,E1 211.799} C_DIS
LIN {X 0.154,Y -432.036,Z 1341.967,A 0.000,B 0.000,C 90.000,E1 210.001} C_DIS
LIN {X 0.041,Y -445.022,Z 1341.962,A 0.000,B 0.000,C 90.000,E1 209.077} C_DIS
LIN {X 0.150,Y -446.302,Z 1341.961,A 0.000,B 0.000,C 90.000,E1 208.949} C_DIS
LIN {X 0.042,Y -447.969,Z 1341.959,A 0.000,B 0.000,C 90.000,E1 208.693} C_DIS
LIN {X 0.107,Y -449.317,Z 1341.958,A 0.000,B 0.000,C 90.000,E1 208.359} C_DIS
LIN {X 0.181,Y -450.354,Z 1341.956,A 0.000,B 0.000,C 90.000,E1 208.025} C_DIS
LIN {X 0.126,Y -451.947,Z 1341.952,A 0.000,B 0.000,C 90.000,E1 207.385} C_DIS
LIN {X 0.087,Y -453.107,Z 1341.949,A 0.000,B 0.000,C 90.000,E1 206.744} C_DIS
LIN {X -0.074,Y -455.344,Z 1341.940,A 0.000,B 0.000,C 90.000,E1 205.155} C_DIS
LIN {X 0.221,Y -457.450,Z 1341.931,A 0.000,B 0.000,C 90.000,E1 203.515} C_DIS
LIN {X -0.055,Y -459.407,Z 1341.922,A 0.000,B 0.000,C 90.000,E1 201.950} C_DIS
LIN {X 0.036,Y -461.023,Z 1341.915,A 0.000,B 0.000,C 90.000,E1 200.663} C_DIS
LIN {X 0.210,Y -463.648,Z 1341.902,A 0.000,B 0.000,C 90.000,E1 198.417} C_DIS
LIN {X -0.072,Y -465.806,Z 1341.892,A 0.000,B 0.000,C 90.000,E1 196.551} C_DIS
LIN {X 0.074,Y -468.289,Z 1341.878,A 0.000,B 0.000,C 90.000,E1 194.008} C_DIS
LIN {X 0.093,Y -470.176,Z 1341.867,A 0.000,B 0.000,C 90.000,E1 192.119} C_DIS
LIN {X -0.046,Y -472.141,Z 1341.857,A 0.000,B 0.000,C 90.000,E1 190.254} C_DIS
LIN {X 0.024,Y -473.670,Z 1341.848,A 0.000,B 0.000,C 90.000,E1 188.681} C_DIS
LIN {X 0.213,Y -474.777,Z 1341.841,A 0.000,B 0.000,C 90.000,E1 187.409} C_DIS
LIN {X 0.116,Y -475.556,Z 1341.836,A 0.000,B 0.000,C 90.000,E1 186.486} C_DIS
LIN {X -0.194,Y -476.255,Z 1341.829,A 0.000,B 0.000,C 90.000,E1 185.277} C_DIS
LIN {X 0.156,Y -476.785,Z 1341.824,A 0.000,B 0.000,C 90.000,E1 184.302} C_DIS
LIN {X 0.132,Y -477.238,Z 1341.815,A 0.000,B 0.000,C 90.000,E1 182.751} C_DIS
LIN {X 0.087,Y -477.209,Z 1341.807,A 0.000,B 0.000,C 90.000,E1 181.203} C_DIS
LIN {X -0.042,Y -476.951,Z 1341.802,A 0.000,B 0.000,C 90.000,E1 180.286} C_DIS
LIN {X -0.172,Y -476.522,Z 1341.796,A 0.000,B 0.000,C 90.000,E1 179.370} C_DIS
LIN {X -0.025,Y -475.693,Z 1341.790,A 0.000,B 0.000,C 90.000,E1 178.108} C_DIS
LIN {X 0.113,Y -474.538,Z 1341.783,A 0.000,B 0.000,C 90.000,E1 176.846} C_DIS
LIN {X -0.024,Y -473.448,Z 1341.777,A 0.000,B 0.000,C 90.000,E1 175.927} C_DIS
LIN {X -0.177,Y -472.012,Z 1341.772,A 0.000,B 0.000,C 90.000,E1 175.008} C_DIS
LIN {X -0.118,Y -470.958,Z 1341.769,A 0.000,B 0.000,C 90.000,E1 174.375} C_DIS
LIN {X -0.068,Y -469.569,Z 1341.765,A 0.000,B 0.000,C 90.000,E1 173.742} C_DIS
LIN {X -0.219,Y -466.873,Z 1341.760,A 0.000,B 0.000,C 90.000,E1 172.818} C_DIS
LIN {X -0.204,Y -464.698,Z 1341.756,A 0.000,B 0.000,C 90.000,E1 172.186} C_DIS
LIN {X 0.107,Y -460.483,Z 1341.751,A 0.000,B 0.000,C 90.000,E1 171.197} C_DIS
LIN {X -0.103,Y -458.899,Z 1341.750,A 0.000,B 0.000,C 90.000,E1 170.905} C_DIS
LIN {X -0.011,Y -454.512,Z 1341.745,A 0.000,B 0.000,C 90.000,E1 170.095} C_DIS
LIN {X 0.173,Y -448.542,Z 1341.740,A 0.000,B 0.000,C 90.000,E1 169.106} C_DIS
LIN {X -0.154,Y -442.154,Z 1341.734,A 0.000,B 0.000,C 90.000,E1 168.173} C_DIS
LIN {X 0.104,Y -433.390,Z 1341.727,A 0.000,B 0.000,C 90.000,E1 166.825} C_DIS
LIN {X 0.164,Y -420.380,Z 1341.716,A 0.000,B 0.000,C 90.000,E1 164.810} C_DIS
LIN {X -0.016,Y -416.436,Z 1341.712,A 0.000,B 0.000,C 90.000,E1 164.157} C_DIS
LIN {X 0.140,Y -414.839,Z 1341.710,A 0.000,B 0.000,C 90.000,E1 163.795} C_DIS
LIN {X -0.152,Y -413.060,Z 1341.707,A 0.000,B 0.000,C 90.000,E1 163.323} C_DIS
LIN {X 0.105,Y -412.509,Z 1341.705,A 0.000,B 0.000,C 90.000,E1 162.960} C_DIS
LIN {X -0.030,Y -412.511,Z 1341.705,A 0.000,B 0.000,C 90.000,E1 162.834} C_DIS
LIN {X 0.023,Y -413.672,Z 1341.703,A 0.000,B 0.000,C 90.000,E1 162.489} C_DIS
LIN {X -0.016,Y -413.703,Z 1341.703,A 0.000,B 0.000,C 90.000,E1 162.489} C_DIS
LIN {X -0.120,Y -416.521,Z 1341.701,A 0.000,B 0.000,C 90.000,E1 162.127} C_DIS
LIN {X 0.186,Y -422.691,Z 1341.697,A 0.000,B 0.000,C 90.000,E1 161.456} C_DIS
LIN {X 0.103,Y -431.422,Z 1341.693,A 0.000,B 0.000,C 90.000,E1 160.732} C_DIS
LIN {X 0.044,Y -445.730,Z 1341.687,A 0.000,B 0.000,C 90.000,E1 159.645} C_DIS
LIN {X -0.122,Y -458.223,Z 1341.682,A 0.000,B 0.000,C 90.000,E1 158.720} C_DIS
LIN {X -0.044,Y -464.445,Z 1341.679,A 0.000,B 0.000,C 90.000,E1 158.230} C_DIS
LIN {X 0.029,Y -475.114,Z 1341.674,A 0.000,B 0.000,C 90.000,E1 157.358} C_DIS
LIN {X -0.074,Y -482.477,Z 1341.671,A 0.000,B 0.000,C 90.000,E1 156.741} C_DIS
LIN {X -0.119,Y -488.230,Z 1341.668,A 0.000,B 0.000,C 90.000,E1 156.230} C_DIS
LIN {X 0.085,Y -495.234,Z 1341.664,A 0.000,B 0.000,C 90.000,E1 155.537} C_DIS
LIN {X 0.237,Y -500.728,Z 1341.661,A 0.000,B 0.000,C 90.000,E1 154.973} C_DIS
LIN {X 0.134,Y -507.430,Z 1341.657,A 0.000,B 0.000,C 90.000,E1 154.280} C_DIS
LIN {X -0.131,Y -513.875,Z 1341.653,A 0.000,B 0.000,C 90.000,E1 153.589} C_DIS
LIN {X 0.038,Y -517.544,Z 1341.651,A 0.000,B 0.000,C 90.000,E1 153.127} C_DIS
LIN {X -0.019,Y -522.973,Z 1341.647,A 0.000,B 0.000,C 90.000,E1 152.410} C_DIS
LIN {X -0.036,Y -526.052,Z 1341.644,A 0.000,B 0.000,C 90.000,E1 151.975} C_DIS
LIN {X 0.056,Y -529.655,Z 1341.641,A 0.000,B 0.000,C 90.000,E1 151.385} C_DIS
LIN {X 0.028,Y -533.234,Z 1341.637,A 0.000,B 0.000,C 90.000,E1 150.667} C_DIS
LIN {X 0.174,Y -535.666,Z 1341.634,A 0.000,B 0.000,C 90.000,E1 150.078} C_DIS
LIN {X -0.128,Y -537.715,Z 1341.631,A 0.000,B 0.000,C 90.000,E1 149.537} C_DIS
LIN {X 0.048,Y -540.367,Z 1341.626,A 0.000,B 0.000,C 90.000,E1 148.663} C_DIS
LIN {X -0.220,Y -541.995,Z 1341.623,A 0.000,B 0.000,C 90.000,E1 148.122} C_DIS
LIN {X 0.004,Y -544.031,Z 1341.618,A 0.000,B 0.000,C 90.000,E1 147.248} C_DIS
LIN {X -0.208,Y -545.742,Z 1341.613,A 0.000,B 0.000,C 90.000,E1 146.421} C_DIS
LIN {X 0.049,Y -547.200,Z 1341.609,A 0.000,B 0.000,C 90.000,E1 145.548} C_DIS
LIN {X 0.134,Y -547.994,Z 1341.606,A 0.000,B 0.000,C 90.000,E1 144.975} C_DIS
LIN {X 0.006,Y -549.306,Z 1341.599,A 0.000,B 0.000,C 90.000,E1 143.863} C_DIS
LIN {X -0.220,Y -550.268,Z 1341.593,A 0.000,B 0.000,C 90.000,E1 142.763} C_DIS
LIN {X 0.067,Y -551.177,Z 1341.585,A 0.000,B 0.000,C 90.000,E1 141.331} C_DIS
LIN {X -0.082,Y -552.266,Z 1341.576,A 0.000,B 0.000,C 90.000,E1 139.666} C_DIS
LIN {X 0.285,Y -553.735,Z 1341.563,A 0.000,B 0.000,C 90.000,E1 137.391} C_DIS
LIN {X 0.018,Y -554.509,Z 1341.559,A 0.000,B 0.000,C 90.000,E1 136.581} C_DIS
LIN {X 0.289,Y -554.919,Z 1341.557,A 0.000,B 0.000,C 90.000,E1 136.134} C_DIS
LIN {X -0.058,Y -555.817,Z 1341.555,A 0.000,B 0.000,C 90.000,E1 135.891} C_DIS
LIN {X -0.286,Y -556.019,Z 1341.554,A 0.000,B 0.000,C 90.000,E1 135.810} C_DIS
LIN {X -0.328,Y -556.041,Z 1341.554,A 0.000,B 0.000,C 90.000,E1 135.810} C_DIS
LIN {X 0.162,Y -556.430,Z 1341.554,A 0.000,B 0.000,C 90.000,E1 135.729} C_DIS
LIN {X -0.298,Y -558.979,Z 1341.553,A 0.000,B 0.000,C 90.000,E1 135.486} C_DIS
LIN {X -0.285,Y -570.386,Z 1341.551,A 0.000,B 0.000,C 90.000,E1 135.162} C_DIS
LIN {X -0.074,Y -573.552,Z 1341.550,A 0.000,B 0.000,C 90.000,E1 135.040} C_DIS
LIN {X 0.029,Y -576.165,Z 1341.550,A 0.000,B 0.000,C 90.000,E1 134.919} C_DIS
LIN {X 0.208,Y -579.164,Z 1341.549,A 0.000,B 0.000,C 90.000,E1 134.757} C_DIS
LIN {X 0.234,Y -582.135,Z 1341.548,A 0.000,B 0.000,C 90.000,E1 134.595} C_DIS
LIN {X -0.180,Y -588.230,Z 1341.546,A 0.000,B 0.000,C 90.000,E1 134.271} C_DIS
LIN {X -0.067,Y -593.875,Z 1341.544,A 0.000,B 0.000,C 90.000,E1 133.866} C_DIS
LIN {X 0.116,Y -600.504,Z 1341.541,A 0.000,B 0.000,C 90.000,E1 133.299} C_DIS
LIN {X -0.196,Y -605.745,Z 1341.538,A 0.000,B 0.000,C 90.000,E1 132.852} C_DIS
LIN {X 0.086,Y -611.966,Z 1341.535,A 0.000,B 0.000,C 90.000,E1 132.204} C_DIS
LIN {X -0.059,Y -617.541,Z 1341.531,A 0.000,B 0.000,C 90.000,E1 131.595} C_DIS
LIN {X 0.083,Y -621.988,Z 1341.528,A 0.000,B 0.000,C 90.000,E1 131.067} C_DIS
LIN {X -0.257,Y -627.204,Z 1341.525,A 0.000,B 0.000,C 90.000,E1 130.458} C_DIS
LIN {X -0.072,Y -632.207,Z 1341.521,A 0.000,B 0.000,C 90.000,E1 129.806} C_DIS
LIN {X 0.101,Y -637.854,Z 1341.517,A 0.000,B 0.000,C 90.000,E1 129.036} C_DIS
LIN {X -0.118,Y -643.206,Z 1341.513,A 0.000,B 0.000,C 90.000,E1 128.302} C_DIS
LIN {X 0.209,Y -647.560,Z 1341.509,A 0.000,B 0.000,C 90.000,E1 127.649} C_DIS
LIN {X -0.012,Y -653.302,Z 1341.505,A 0.000,B 0.000,C 90.000,E1 126.824} C_DIS
LIN {X -0.084,Y -657.977,Z 1341.500,A 0.000,B 0.000,C 90.000,E1 126.091} C_DIS
LIN {X -0.014,Y -661.659,Z 1341.497,A 0.000,B 0.000,C 90.000,E1 125.471} C_DIS
LIN {X -0.071,Y -663.076,Z 1341.496,A 0.000,B 0.000,C 90.000,E1 125.231} C_DIS
LIN {X 0.102,Y -666.814,Z 1341.492,A 0.000,B 0.000,C 90.000,E1 124.485} C_DIS
LIN {X 0.182,Y -669.130,Z 1341.489,A 0.000,B 0.000,C 90.000,E1 123.992} C_DIS
LIN {X -0.142,Y -672.207,Z 1341.485,A 0.000,B 0.000,C 90.000,E1 123.293} C_DIS
LIN {X 0.122,Y -674.816,Z 1341.481,A 0.000,B 0.000,C 90.000,E1 122.546} C_DIS
LIN {X 0.415,Y -677.078,Z 1341.477,A 0.000,B 0.000,C 90.000,E1 121.799} C_DIS
LIN {X -0.203,Y -679.081,Z 1341.473,A 0.000,B 0.000,C 90.000,E1 121.131} C_DIS
LIN {X 0.127,Y -680.793,Z 1341.469,A 0.000,B 0.000,C 90.000,E1 120.384} C_DIS
LIN {X 0.129,Y -682.140,Z 1341.465,A 0.000,B 0.000,C 90.000,E1 119.667} C_DIS
LIN {X 0.148,Y -683.113,Z 1341.461,A 0.000,B 0.000,C 90.000,E1 118.949} C_DIS
LIN {X -0.003,Y -683.871,Z 1341.454,A 0.000,B 0.000,C 90.000,E1 117.769} C_DIS
LIN {X 0.030,Y -683.932,Z 1341.450,A 0.000,B 0.000,C 90.000,E1 117.052} C_DIS
LIN {X -0.033,Y -683.715,Z 1341.445,A 0.000,B 0.000,C 90.000,E1 116.104} C_DIS
LIN {X -0.305,Y -683.232,Z 1341.441,A 0.000,B 0.000,C 90.000,E1 115.412} C_DIS
LIN {X 0.120,Y -682.691,Z 1341.438,A 0.000,B 0.000,C 90.000,E1 114.899} C_DIS
LIN {X -0.367,Y -681.717,Z 1341.436,A 0.000,B 0.000,C 90.000,E1 114.463} C_DIS
LIN {X -0.160,Y -681.138,Z 1341.434,A 0.000,B 0.000,C 90.000,E1 114.207} C_DIS
LIN {X 0.243,Y -679.305,Z 1341.432,A 0.000,B 0.000,C 90.000,E1 113.695} C_DIS
LIN {X 0.070,Y -678.759,Z 1341.431,A 0.000,B 0.000,C 90.000,E1 113.590} C_DIS
LIN {X 0.264,Y -676.894,Z 1341.430,A 0.000,B 0.000,C 90.000,E1 113.334} C_DIS
LIN {X -0.079,Y -673.849,Z 1341.428,A 0.000,B 0.000,C 90.000,E1 113.003} C_DIS
LIN {X -0.253,Y -672.262,Z 1341.427,A 0.000,B 0.000,C 90.000,E1 112.898} C_DIS
LIN {X -0.099,Y -665.399,Z 1341.425,A 0.000,B 0.000,C 90.000,E1 112.514} C_DIS
LIN {X 0.193,Y -663.504,Z 1341.425,A 0.000,B 0.000,C 90.000,E1 112.408} C_DIS
LIN {X 0.042,Y -659.077,Z 1341.424,A 0.000,B 0.000,C 90.000,E1 112.280} C_DIS
LIN {X 0.285,Y -656.756,Z 1341.424,A 0.000,B 0.000,C 90.000,E1 112.206} C_DIS
LIN {X 0.086,Y -639.372,Z 1341.422,A 0.000,B 0.000,C 90.000,E1 111.897} C_DIS
LIN {X 0.040,Y -639.348,Z 1341.422,A 0.000,B 0.000,C 90.000,E1 111.897} C_DIS
LIN {X 0.171,Y -641.509,Z 1341.420,A 0.000,B 0.000,C 90.000,E1 111.589} C_DIS
LIN {X -0.242,Y -647.330,Z 1341.416,A 0.000,B 0.000,C 90.000,E1 110.918} C_DIS
LIN {X -0.328,Y -651.116,Z 1341.413,A 0.000,B 0.000,C 90.000,E1 110.429} C_DIS
LIN {X 0.270,Y -655.099,Z 1341.410,A 0.000,B 0.000,C 90.000,E1 109.758} C_DIS
LIN {X 0.236,Y -657.859,Z 1341.407,A 0.000,B 0.000,C 90.000,E1 109.268} C_DIS
LIN {X 0.055,Y -660.882,Z 1341.404,A 0.000,B 0.000,C 90.000,E1 108.671} C_DIS
LIN {X -0.047,Y -664.057,Z 1341.400,A 0.000,B 0.000,C 90.000,E1 107.946} C_DIS
LIN {X -0.121,Y -666.911,Z 1341.396,A 0.000,B 0.000,C 90.000,E1 107.221} C_DIS
LIN {X -0.172,Y -669.456,Z 1341.392,A 0.000,B 0.000,C 90.000,E1 106.496} C_DIS
LIN {X -0.319,Y -670.988,Z 1341.389,A 0.000,B 0.000,C 90.000,E1 106.024} C_DIS
LIN {X 0.309,Y -672.937,Z 1341.385,A 0.000,B 0.000,C 90.000,E1 105.245} C_DIS
LIN {X 0.131,Y -674.550,Z 1341.381,A 0.000,B 0.000,C 90.000,E1 104.537} C_DIS
LIN {X 0.023,Y -675.399,Z 1341.378,A 0.000,B 0.000,C 90.000,E1 104.064} C_DIS
LIN {X -0.081,Y -676.075,Z 1341.375,A 0.000,B 0.000,C 90.000,E1 103.592} C_DIS
LIN {X -0.181,Y -676.551,Z 1341.373,A 0.000,B 0.000,C 90.000,E1 103.119} C_DIS
LIN {X -0.279,Y -676.787,Z 1341.370,A 0.000,B 0.000,C 90.000,E1 102.647} C_DIS
LIN {X 0.095,Y -676.799,Z 1341.366,A 0.000,B 0.000,C 90.000,E1 101.895} C_DIS
LIN {X -0.001,Y -676.635,Z 1341.364,A 0.000,B 0.000,C 90.000,E1 101.422} C_DIS
LIN {X -0.103,Y -676.226,Z 1341.361,A 0.000,B 0.000,C 90.000,E1 100.950} C_DIS
LIN {X -0.334,Y -675.604,Z 1341.358,A 0.000,B 0.000,C 90.000,E1 100.489} C_DIS
LIN {X 0.159,Y -674.247,Z 1341.354,A 0.000,B 0.000,C 90.000,E1 99.726} C_DIS
LIN {X -0.079,Y -673.041,Z 1341.351,A 0.000,B 0.000,C 90.000,E1 99.265} C_DIS
LIN {X -0.319,Y -671.475,Z 1341.349,A 0.000,B 0.000,C 90.000,E1 98.803} C_DIS
LIN {X 0.017,Y -668.601,Z 1341.345,A 0.000,B 0.000,C 90.000,E1 98.049} C_DIS
LIN {X 0.320,Y -665.364,Z 1341.341,A 0.000,B 0.000,C 90.000,E1 97.296} C_DIS
LIN {X -0.171,Y -661.076,Z 1341.336,A 0.000,B 0.000,C 90.000,E1 96.486} C_DIS
LIN {X 0.170,Y -658.398,Z 1341.333,A 0.000,B 0.000,C 90.000,E1 95.967} C_DIS
LIN {X 0.283,Y -653.962,Z 1341.329,A 0.000,B 0.000,C 90.000,E1 95.220} C_DIS
LIN {X -0.027,Y -651.589,Z 1341.327,A 0.000,B 0.000,C 90.000,E1 94.878} C_DIS
LIN {X 0.247,Y -648.209,Z 1341.324,A 0.000,B 0.000,C 90.000,E1 94.359} C_DIS
LIN {X -0.152,Y -644.648,Z 1341.322,A 0.000,B 0.000,C 90.000,E1 93.898} C_DIS
LIN {X 0.028,Y -640.801,Z 1341.319,A 0.000,B 0.000,C 90.000,E1 93.383} C_DIS
LIN {X 0.092,Y -635.153,Z 1341.315,A 0.000,B 0.000,C 90.000,E1 92.751} C_DIS
LIN {X 0.250,Y -628.924,Z 1341.312,A 0.000,B 0.000,C 90.000,E1 92.121} C_DIS
LIN {X 0.265,Y -618.965,Z 1341.307,A 0.000,B 0.000,C 90.000,E1 91.146} C_DIS
LIN {X -0.011,Y -614.752,Z 1341.304,A 0.000,B 0.000,C 90.000,E1 90.802} C_DIS
LIN {X 0.016,Y -609.324,Z 1341.302,A 0.000,B 0.000,C 90.000,E1 90.344} C_DIS
LIN {X -0.069,Y -602.900,Z 1341.300,A 0.000,B 0.000,C 90.000,E1 89.943} C_DIS
LIN {X -0.169,Y -595.994,Z 1341.298,A 0.000,B 0.000,C 90.000,E1 89.599} C_DIS
LIN {X 0.256,Y -588.919,Z 1341.296,A 0.000,B 0.000,C 90.000,E1 89.255} C_DIS
LIN {X 0.256,Y -580.641,Z 1341.294,A 0.000,B 0.000,C 90.000,E1 88.912} C_DIS
LIN {X 0.106,Y -577.829,Z 1341.293,A 0.000,B 0.000,C 90.000,E1 88.797} C_DIS
LIN {X -0.087,Y -576.610,Z 1341.293,A 0.000,B 0.000,C 90.000,E1 88.740} C_DIS
LIN {X 0.179,Y -573.470,Z 1341.292,A 0.000,B 0.000,C 90.000,E1 88.453} C_DIS
LIN {X -0.186,Y -573.178,Z 1341.291,A 0.000,B 0.000,C 90.000,E1 88.453} C_DIS
LIN {X -0.223,Y -573.156,Z 1341.291,A 0.000,B 0.000,C 90.000,E1 88.453} C_DIS
LIN {X -0.050,Y -572.575,Z 1341.290,A 0.000,B 0.000,C 90.000,E1 88.165} C_DIS
LIN {X 0.146,Y -572.648,Z 1341.287,A 0.000,B 0.000,C 90.000,E1 87.593} C_DIS
LIN {X 0.172,Y -574.655,Z 1341.275,A 0.000,B 0.000,C 90.000,E1 85.412} C_DIS
LIN {X -0.227,Y -577.068,Z 1341.263,A 0.000,B 0.000,C 90.000,E1 83.280} C_DIS
LIN {X 0.311,Y -579.018,Z 1341.254,A 0.000,B 0.000,C 90.000,E1 81.602} C_DIS
LIN {X 0.088,Y -580.677,Z 1341.246,A 0.000,B 0.000,C 90.000,E1 80.274} C_DIS
LIN {X 0.323,Y -582.457,Z 1341.237,A 0.000,B 0.000,C 90.000,E1 78.634} C_DIS
LIN {X -0.329,Y -583.696,Z 1341.230,A 0.000,B 0.000,C 90.000,E1 77.353} C_DIS
LIN {X -0.137,Y -584.854,Z 1341.222,A 0.000,B 0.000,C 90.000,E1 75.992} C_DIS
LIN {X 0.083,Y -585.850,Z 1341.215,A 0.000,B 0.000,C 90.000,E1 74.629} C_DIS
LIN {X 0.158,Y -586.955,Z 1341.206,A 0.000,B 0.000,C 90.000,E1 73.015} C_DIS
LIN {X 0.015,Y -587.756,Z 1341.198,A 0.000,B 0.000,C 90.000,E1 71.692} C_DIS
LIN {X 0.304,Y -588.791,Z 1341.189,A 0.000,B 0.000,C 90.000,E1 70.061} C_DIS
LIN {X -0.193,Y -590.091,Z 1341.178,A 0.000,B 0.000,C 90.000,E1 67.975} C_DIS
LIN {X 0.008,Y -591.216,Z 1341.169,A 0.000,B 0.000,C 90.000,E1 66.357} C_DIS
LIN {X 0.120,Y -592.578,Z 1341.158,A 0.000,B 0.000,C 90.000,E1 64.485} C_DIS
LIN {X -0.196,Y -593.672,Z 1341.150,A 0.000,B 0.000,C 90.000,E1 62.922} C_DIS
LIN {X -0.128,Y -595.442,Z 1341.138,A 0.000,B 0.000,C 90.000,E1 60.795} C_DIS
LIN {X -0.200,Y -596.472,Z 1341.132,A 0.000,B 0.000,C 90.000,E1 59.744} C_DIS
LIN {X 0.177,Y -598.051,Z 1341.123,A 0.000,B 0.000,C 90.000,E1 58.122} C_DIS
LIN {X 0.091,Y -599.640,Z 1341.114,A 0.000,B 0.000,C 90.000,E1 56.548} C_DIS
LIN {X 0.032,Y -601.242,Z 1341.105,A 0.000,B 0.000,C 90.000,E1 54.975} C_DIS
LIN {X 0.083,Y -602.471,Z 1341.098,A 0.000,B 0.000,C 90.000,E1 53.657} C_DIS
LIN {X -0.232,Y -603.487,Z 1341.092,A 0.000,B 0.000,C 90.000,E1 52.637} C_DIS
LIN {X 0.321,Y -604.245,Z 1341.087,A 0.000,B 0.000,C 90.000,E1 51.537} C_DIS
LIN {X -0.171,Y -605.151,Z 1341.079,A 0.000,B 0.000,C 90.000,E1 50.275} C_DIS
LIN {X -0.057,Y -605.720,Z 1341.073,A 0.000,B 0.000,C 90.000,E1 49.218} C_DIS
LIN {X 0.064,Y -606.113,Z 1341.068,A 0.000,B 0.000,C 90.000,E1 48.162} C_DIS
LIN {X -0.070,Y -606.269,Z 1341.063,A 0.000,B 0.000,C 90.000,E1 47.391} C_DIS
LIN {X 0.078,Y -606.493,Z 1341.055,A 0.000,B 0.000,C 90.000,E1 45.810} C_DIS
LIN {X 0.176,Y -606.475,Z 1341.049,A 0.000,B 0.000,C 90.000,E1 44.757} C_DIS
LIN {X 0.272,Y -606.258,Z 1341.043,A 0.000,B 0.000,C 90.000,E1 43.704} C_DIS
LIN {X 0.004,Y -605.640,Z 1341.034,A 0.000,B 0.000,C 90.000,E1 42.162} C_DIS
LIN {X -0.074,Y -605.067,Z 1341.027,A 0.000,B 0.000,C 90.000,E1 40.862} C_DIS
LIN {X 0.040,Y -604.561,Z 1341.021,A 0.000,B 0.000,C 90.000,E1 39.806} C_DIS
LIN {X -0.191,Y -603.776,Z 1341.012,A 0.000,B 0.000,C 90.000,E1 38.257} C_DIS
LIN {X 0.364,Y -602.906,Z 1341.007,A 0.000,B 0.000,C 90.000,E1 37.156} C_DIS
LIN {X 0.053,Y -601.729,Z 1341.001,A 0.000,B 0.000,C 90.000,E1 36.137} C_DIS
LIN {X -0.141,Y -600.042,Z 1340.995,A 0.000,B 0.000,C 90.000,E1 35.105} C_DIS
LIN {X -0.249,Y -598.607,Z 1340.991,A 0.000,B 0.000,C 90.000,E1 34.326} C_DIS
LIN {X 0.021,Y -596.487,Z 1340.985,A 0.000,B 0.000,C 90.000,E1 33.245} C_DIS
LIN {X -0.352,Y -595.298,Z 1340.982,A 0.000,B 0.000,C 90.000,E1 32.752} C_DIS
LIN {X -0.125,Y -592.573,Z 1340.976,A 0.000,B 0.000,C 90.000,E1 31.671} C_DIS
LIN {X 0.058,Y -589.155,Z 1340.970,A 0.000,B 0.000,C 90.000,E1 30.590} C_DIS
LIN {X 0.012,Y -586.318,Z 1340.966,A 0.000,B 0.000,C 90.000,E1 29.795} C_DIS
LIN {X -0.064,Y -582.951,Z 1340.961,A 0.000,B 0.000,C 90.000,E1 28.999} C_DIS
LIN {X 0.189,Y -580.606,Z 1340.958,A 0.000,B 0.000,C 90.000,E1 28.437} C_DIS
LIN {X 0.193,Y -578.042,Z 1340.955,A 0.000,B 0.000,C 90.000,E1 27.897} C_DIS
LIN {X -0.174,Y -574.510,Z 1340.951,A 0.000,B 0.000,C 90.000,E1 27.257} C_DIS
LIN {X -0.051,Y -570.794,Z 1340.948,A 0.000,B 0.000,C 90.000,E1 26.565} C_DIS
LIN {X 0.289,Y -566.723,Z 1340.944,A 0.000,B 0.000,C 90.000,E1 25.848} C_DIS
LIN {X -0.168,Y -562.225,Z 1340.940,A 0.000,B 0.000,C 90.000,E1 25.207} C_DIS
LIN {X -0.155,Y -557.386,Z 1340.936,A 0.000,B 0.000,C 90.000,E1 24.515} C_DIS
LIN {X 0.038,Y -554.339,Z 1340.934,A 0.000,B 0.000,C 90.000,E1 24.079} C_DIS
LIN {X -0.137,Y -547.914,Z 1340.929,A 0.000,B 0.000,C 90.000,E1 23.259} C_DIS
LIN {X 0.247,Y -542.061,Z 1340.925,A 0.000,B 0.000,C 90.000,E1 22.514} C_DIS
LIN {X -0.127,Y -533.684,Z 1340.920,A 0.000,B 0.000,C 90.000,E1 21.589} C_DIS
LIN {X -0.016,Y -523.487,Z 1340.914,A 0.000,B 0.000,C 90.000,E1 20.482} C_DIS
LIN {X -0.220,Y -512.942,Z 1340.908,A 0.000,B 0.000,C 90.000,E1 19.396} C_DIS
LIN {X 0.206,Y -503.664,Z 1340.902,A 0.000,B 0.000,C 90.000,E1 18.362} C_DIS
LIN {X -0.136,Y -493.042,Z 1340.896,A 0.000,B 0.000,C 90.000,E1 17.330} C_DIS
LIN {X -0.145,Y -481.515,Z 1340.890,A 0.000,B 0.000,C 90.000,E1 16.260} C_DIS
LIN {X -0.068,Y -471.521,Z 1340.885,A 0.000,B 0.000,C 90.000,E1 15.300} C_DIS
LIN {X 0.190,Y -461.400,Z 1340.880,A 0.000,B 0.000,C 90.000,E1 14.300} C_DIS
LIN {X -0.041,Y -448.442,Z 1340.873,A 0.000,B 0.000,C 90.000,E1 13.063} C_DIS
LIN {X 0.054,Y -427.041,Z 1340.860,A 0.000,B 0.000,C 90.000,E1 10.838} C_DIS
LIN {X 0.059,Y -414.424,Z 1340.853,A 0.000,B 0.000,C 90.000,E1 9.443} C_DIS
LIN {X 0.194,Y -405.921,Z 1340.847,A 0.000,B 0.000,C 90.000,E1 8.454} C_DIS
LIN {X 0.063,Y -397.877,Z 1340.842,A 0.000,B 0.000,C 90.000,E1 7.530} C_DIS
LIN {X -0.005,Y -395.943,Z 1340.841,A 0.000,B 0.000,C 90.000,E1 7.296} C_DIS
LIN {X 0.088,Y -394.941,Z 1340.839,A 0.000,B 0.000,C 90.000,E1 7.068} C_DIS
LIN {X 0.051,Y -394.920,Z 1340.839,A 0.000,B 0.000,C 90.000,E1 7.068} C_DIS
LIN {X 0.138,Y -394.953,Z 1340.839,A 0.000,B 0.000,C 90.000,E1 7.011} C_DIS
LIN {X 0.100,Y -394.975,Z 1340.839,A 0.000,B 0.000,C 90.000,E1 7.011} C_DIS
LIN {X 0.009,Y -395.569,Z 1340.839,A 0.000,B 0.000,C 90.000,E1 6.947} C_DIS
LIN {X -0.191,Y -399.781,Z 1340.837,A 0.000,B 0.000,C 90.000,E1 6.606} C_DIS
LIN {X -0.067,Y -408.726,Z 1340.833,A 0.000,B 0.000,C 90.000,E1 5.967} C_DIS
LIN {X 0.027,Y -416.939,Z 1340.830,A 0.000,B 0.000,C 90.000,E1 5.391} C_DIS
LIN {X -0.200,Y -423.135,Z 1340.827,A 0.000,B 0.000,C 90.000,E1 4.935} C_DIS
LIN {X 0.113,Y -429.146,Z 1340.824,A 0.000,B 0.000,C 90.000,E1 4.359} C_DIS
LIN {X -0.056,Y -436.345,Z 1340.820,A 0.000,B 0.000,C 90.000,E1 3.669} C_DIS
LIN {X -0.181,Y -442.089,Z 1340.817,A 0.000,B 0.000,C 90.000,E1 3.094} C_DIS
LIN {X 0.099,Y -448.928,Z 1340.813,A 0.000,B 0.000,C 90.000,E1 2.293} C_DIS
LIN {X 0.180,Y -454.339,Z 1340.809,A 0.000,B 0.000,C 90.000,E1 1.661} C_DIS
LIN {X 0.230,Y -460.773,Z 1340.805,A 0.000,B 0.000,C 90.000,E1 0.859} C_DIS
LIN {X 0.000,Y -467.316,Z 1340.800,A 0.000,B 0.000,C 90.000,E1 360.000} C_DIS
LIN {X 0.064,Y -472.086,Z 1340.796,A 0.000,B 0.000,C 90.000,E1 359.312} C_DIS
LIN {X 0.229,Y -477.072,Z 1340.792,A 0.000,B 0.000,C 90.000,E1 358.511} C_DIS
LIN {X -0.020,Y -481.739,Z 1340.788,A 0.000,B 0.000,C 90.000,E1 357.764} C_DIS
LIN {X -0.250,Y -486.030,Z 1340.783,A 0.000,B 0.000,C 90.000,E1 357.020} C_DIS
LIN {X -0.090,Y -489.306,Z 1340.780,A 0.000,B 0.000,C 90.000,E1 356.388} C_DIS
LIN {X -0.224,Y -492.959,Z 1340.776,A 0.000,B 0.000,C 90.000,E1 355.641} C_DIS
LIN {X -0.154,Y -496.986,Z 1340.771,A 0.000,B 0.000,C 90.000,E1 354.723} C_DIS
LIN {X -0.170,Y -500.135,Z 1340.766,A 0.000,B 0.000,C 90.000,E1 353.970} C_DIS
LIN {X -0.028,Y -503.641,Z 1340.761,A 0.000,B 0.000,C 90.000,E1 353.053} C_DIS
LIN {X 0.205,Y -506.707,Z 1340.756,A 0.000,B 0.000,C 90.000,E1 352.129} C_DIS
LIN {X 0.094,Y -508.622,Z 1340.753,A 0.000,B 0.000,C 90.000,E1 351.546} C_DIS
LIN {X -0.159,Y -511.835,Z 1340.747,A 0.000,B 0.000,C 90.000,E1 350.387} C_DIS
LIN {X 0.226,Y -514.734,Z 1340.740,A 0.000,B 0.000,C 90.000,E1 349.162} C_DIS
LIN {X 0.167,Y -516.661,Z 1340.735,A 0.000,B 0.000,C 90.000,E1 348.285} C_DIS
LIN {X 0.128,Y -518.415,Z 1340.730,A 0.000,B 0.000,C 90.000,E1 347.409} C_DIS
LIN {X 0.218,Y -520.298,Z 1340.724,A 0.000,B 0.000,C 90.000,E1 346.228} C_DIS
LIN {X -0.298,Y -521.514,Z 1340.719,A 0.000,B 0.000,C 90.000,E1 345.408} C_DIS
LIN {X -0.169,Y -522.465,Z 1340.714,A 0.000,B 0.000,C 90.000,E1 344.519} C_DIS
LIN {X 0.117,Y -523.177,Z 1340.709,A 0.000,B 0.000,C 90.000,E1 343.614} C_DIS
LIN {X -0.236,Y -523.683,Z 1340.704,A 0.000,B 0.000,C 90.000,E1 342.779} C_DIS
LIN {X 0.072,Y -523.847,Z 1340.699,A 0.000,B 0.000,C 90.000,E1 341.873} C_DIS
LIN {X -0.282,Y -523.825,Z 1340.695,A 0.000,B 0.000,C 90.000,E1 341.040} C_DIS
LIN {X 0.021,Y -523.407,Z 1340.690,A 0.000,B 0.000,C 90.000,E1 340.134} C_DIS
LIN {X -0.150,Y -523.026,Z 1340.687,A 0.000,B 0.000,C 90.000,E1 339.571} C_DIS
LIN {X 0.139,Y -522.041,Z 1340.682,A 0.000,B 0.000,C 90.000,E1 338.666} C_DIS
LIN {X -0.036,Y -521.183,Z 1340.678,A 0.000,B 0.000,C 90.000,E1 338.103} C_DIS
LIN {X -0.211,Y -520.101,Z 1340.675,A 0.000,B 0.000,C 90.000,E1 337.539} C_DIS
LIN {X -0.061,Y -519.721,Z 1340.673,A 0.000,B 0.000,C 90.000,E1 337.230} C_DIS
LIN {X -0.101,Y -518.065,Z 1340.669,A 0.000,B 0.000,C 90.000,E1 336.357} C_DIS
LIN {X 0.176,Y -516.554,Z 1340.665,A 0.000,B 0.000,C 90.000,E1 335.741} C_DIS
LIN {X -0.160,Y -515.674,Z 1340.664,A 0.000,B 0.000,C 90.000,E1 335.485} C_DIS
LIN {X -0.201,Y -513.967,Z 1340.661,A 0.000,B 0.000,C 90.000,E1 335.049} C_DIS
LIN {X 0.138,Y -512.551,Z 1340.660,A 0.000,B 0.000,C 90.000,E1 334.717} C_DIS
LIN {X 0.253,Y -510.628,Z 1340.658,A 0.000,B 0.000,C 90.000,E1 334.409} C_DIS
LIN {X 0.078,Y -509.264,Z 1340.657,A 0.000,B 0.000,C 90.000,E1 334.280} C_DIS
LIN {X -0.061,Y -506.904,Z 1340.656,A 0.000,B 0.000,C 90.000,E1 334.152} C_DIS
LIN {X -0.189,Y -479.783,Z 1340.648,A 0.000,B 0.000,C 90.000,E1 332.615} C_DIS
LIN {X 0.030,Y -454.057,Z 1340.639,A 0.000,B 0.000,C 90.000,E1 330.923} C_DIS
LIN {X -0.096,Y -430.350,Z 1340.629,A 0.000,B 0.000,C 90.000,E1 329.203} C_DIS
LIN {X 0.133,Y -408.634,Z 1340.619,A 0.000,B 0.000,C 90.000,E1 327.375} C_DIS
LIN {X 0.024,Y -388.876,Z 1340.609,A 0.000,B 0.000,C 90.000,E1 325.548} C_DIS
LIN {X 0.077,Y -372.065,Z 1340.599,A 0.000,B 0.000,C 90.000,E1 323.783} C_DIS
LIN {X 0.044,Y -372.034,Z 1340.599,A 0.000,B 0.000,C 90.000,E1 323.783} C_DIS
LIN {X -0.091,Y -377.850,Z 1340.565,A 0.000,B 0.000,C 90.000,E1 317.676} C_DIS
LIN {X -0.077,Y -378.243,Z 1340.563,A 0.000,B 0.000,C 90.000,E1 317.310} C_DIS
LIN {X -0.087,Y -383.957,Z 1340.531,A 0.000,B 0.000,C 90.000,E1 311.515} C_DIS
LIN {X -0.001,Y -384.901,Z 1340.527,A 0.000,B 0.000,C 90.000,E1 310.782} C_DIS
LIN {X 0.172,Y -390.628,Z 1340.495,A 0.000,B 0.000,C 90.000,E1 305.025} C_DIS
LIN {X 0.016,Y -391.123,Z 1340.493,A 0.000,B 0.000,C 90.000,E1 304.692} C_DIS
LIN {X -0.067,Y -391.657,Z 1340.489,A 0.000,B 0.000,C 90.000,E1 303.992} C_DIS
LIN {X -0.170,Y -396.843,Z 1340.459,A 0.000,B 0.000,C 90.000,E1 298.693} C_DIS
LIN {X -0.079,Y -397.290,Z 1340.455,A 0.000,B 0.000,C 90.000,E1 297.975} C_DIS
LIN {X 0.010,Y -401.607,Z 1340.426,A 0.000,B 0.000,C 90.000,E1 292.695} C_DIS
LIN {X 0.132,Y -404.670,Z 1340.395,A 0.000,B 0.000,C 90.000,E1 287.094} C_DIS
LIN {X -0.170,Y -404.734,Z 1340.391,A 0.000,B 0.000,C 90.000,E1 286.441} C_DIS
LIN {X 0.123,Y -406.107,Z 1340.364,A 0.000,B 0.000,C 90.000,E1 281.535} C_DIS
LIN {X 0.143,Y -405.955,Z 1340.360,A 0.000,B 0.000,C 90.000,E1 280.838} C_DIS
LIN {X 0.216,Y -405.683,Z 1340.333,A 0.000,B 0.000,C 90.000,E1 275.967} C_DIS
LIN {X 0.148,Y -404.840,Z 1340.326,A 0.000,B 0.000,C 90.000,E1 274.588} C_DIS
LIN {X -0.150,Y -403.488,Z 1340.304,A 0.000,B 0.000,C 90.000,E1 270.802} C_DIS
LIN {X -0.182,Y -403.280,Z 1340.302,A 0.000,B 0.000,C 90.000,E1 270.458} C_DIS
LIN {X 0.002,Y -398.918,Z 1340.271,A 0.000,B 0.000,C 90.000,E1 264.837} C_DIS
LIN {X -0.130,Y -393.098,Z 1340.242,A 0.000,B 0.000,C 90.000,E1 259.567} C_DIS
LIN {X -0.169,Y -392.821,Z 1340.240,A 0.000,B 0.000,C 90.000,E1 259.218} C_DIS
LIN {X -0.078,Y -386.365,Z 1340.214,A 0.000,B 0.000,C 90.000,E1 254.574} C_DIS
LIN {X -0.115,Y -385.255,Z 1340.208,A 0.000,B 0.000,C 90.000,E1 253.504} C_DIS
LIN {X -0.093,Y -384.742,Z 1340.206,A 0.000,B 0.000,C 90.000,E1 253.142} C_DIS
LIN {X 0.133,Y -377.955,Z 1340.182,A 0.000,B 0.000,C 90.000,E1 248.773} C_DIS
LIN {X -0.132,Y -376.218,Z 1340.174,A 0.000,B 0.000,C 90.000,E1 247.358} C_DIS
LIN {X 0.091,Y -374.242,Z 1340.168,A 0.000,B 0.000,C 90.000,E1 246.230} C_DIS
LIN {X -0.108,Y -367.430,Z 1340.144,A 0.000,B 0.000,C 90.000,E1 241.847} C_DIS
LIN {X 0.009,Y -366.020,Z 1340.137,A 0.000,B 0.000,C 90.000,E1 240.717} C_DIS
LIN {X -0.083,Y -359.176,Z 1340.115,A 0.000,B 0.000,C 90.000,E1 236.628} C_DIS
LIN {X -0.065,Y -355.816,Z 1340.100,A 0.000,B 0.000,C 90.000,E1 233.989} C_DIS
LIN {X 0.233,Y -348.776,Z 1340.075,A 0.000,B 0.000,C 90.000,E1 229.380} C_DIS
LIN {X -0.183,Y -346.171,Z 1340.062,A 0.000,B 0.000,C 90.000,E1 227.148} C_DIS
LIN {X -0.174,Y -345.042,Z 1340.057,A 0.000,B 0.000,C 90.000,E1 226.377} C_DIS
LIN {X 0.009,Y -338.572,Z 1340.030,A 0.000,B 0.000,C 90.000,E1 221.310} C_DIS
LIN {X 0.013,Y -338.103,Z 1340.027,A 0.000,B 0.000,C 90.000,E1 220.825} C_DIS
LIN {X -0.005,Y -338.117,Z 1340.027,A 0.000,B 0.000,C 90.000,E1 220.825} C_DIS
LIN {X 0.034,Y -354.585,Z 1340.015,A 0.000,B 0.000,C 90.000,E1 218.624} C_DIS
LIN {X -0.012,Y -372.362,Z 1340.003,A 0.000,B 0.000,C 90.000,E1 216.537} C_DIS
LIN {X 0.125,Y -390.597,Z 1339.992,A 0.000,B 0.000,C 90.000,E1 214.612} C_DIS
LIN {X 0.021,Y -410.792,Z 1339.982,A 0.000,B 0.000,C 90.000,E1 212.752} C_DIS
LIN {X 0.038,Y -432.993,Z 1339.972,A 0.000,B 0.000,C 90.000,E1 210.924} C_DIS
LIN {X 0.037,Y -444.252,Z 1339.967,A 0.000,B 0.000,C 90.000,E1 210.079} C_DIS
LIN {X -0.178,Y -446.627,Z 1339.966,A 0.000,B 0.000,C 90.000,E1 209.873} C_DIS
LIN {X 0.179,Y -448.113,Z 1339.964,A 0.000,B 0.000,C 90.000,E1 209.539} C_DIS
LIN {X 0.247,Y -449.301,Z 1339.963,A 0.000,B 0.000,C 90.000,E1 209.205} C_DIS
LIN {X 0.106,Y -450.236,Z 1339.961,A 0.000,B 0.000,C 90.000,E1 208.899} C_DIS
LIN {X -0.130,Y -451.720,Z 1339.957,A 0.000,B 0.000,C 90.000,E1 208.281} C_DIS
LIN {X -0.175,Y -452.834,Z 1339.953,A 0.000,B 0.000,C 90.000,E1 207.641} C_DIS
LIN {X -0.208,Y -453.706,Z 1339.950,A 0.000,B 0.000,C 90.000,E1 207.001} C_DIS
LIN {X 0.145,Y -456.311,Z 1339.939,A 0.000,B 0.000,C 90.000,E1 205.027} C_DIS
LIN {X -0.144,Y -458.453,Z 1339.930,A 0.000,B 0.000,C 90.000,E1 203.462} C_DIS
LIN {X -0.052,Y -460.829,Z 1339.920,A 0.000,B 0.000,C 90.000,E1 201.535} C_DIS
LIN {X 0.145,Y -462.069,Z 1339.914,A 0.000,B 0.000,C 90.000,E1 200.556} C_DIS
LIN {X -0.082,Y -464.703,Z 1339.902,A 0.000,B 0.000,C 90.000,E1 198.362} C_DIS
LIN {X -0.267,Y -466.543,Z 1339.893,A 0.000,B 0.000,C 90.000,E1 196.804} C_DIS
LIN {X 0.221,Y -468.778,Z 1339.881,A 0.000,B 0.000,C 90.000,E1 194.537} C_DIS
LIN {X -0.131,Y -470.413,Z 1339.872,A 0.000,B 0.000,C 90.000,E1 193.008} C_DIS
LIN {X 0.128,Y -472.712,Z 1339.860,A 0.000,B 0.000,C 90.000,E1 190.782} C_DIS
LIN {X 0.217,Y -474.318,Z 1339.851,A 0.000,B 0.000,C 90.000,E1 189.208} C_DIS
LIN {X -0.048,Y -475.569,Z 1339.844,A 0.000,B 0.000,C 90.000,E1 187.992} C_DIS
LIN {X 0.011,Y -476.890,Z 1339.836,A 0.000,B 0.000,C 90.000,E1 186.429} C_DIS
LIN {X 0.198,Y -477.680,Z 1339.829,A 0.000,B 0.000,C 90.000,E1 185.163} C_DIS
LIN {X -0.080,Y -478.347,Z 1339.822,A 0.000,B 0.000,C 90.000,E1 183.955} C_DIS
LIN {X 0.095,Y -478.722,Z 1339.815,A 0.000,B 0.000,C 90.000,E1 182.694} C_DIS
LIN {X 0.077,Y -478.734,Z 1339.807,A 0.000,B 0.000,C 90.000,E1 181.146} C_DIS
LIN {X 0.163,Y -478.667,Z 1339.803,A 0.000,B 0.000,C 90.000,E1 180.516} C_DIS
LIN {X -0.146,Y -478.231,Z 1339.796,A 0.000,B 0.000,C 90.000,E1 179.312} C_DIS
LIN {X -0.174,Y -477.256,Z 1339.787,A 0.000,B 0.000,C 90.000,E1 177.764} C_DIS
LIN {X -0.013,Y -476.148,Z 1339.781,A 0.000,B 0.000,C 90.000,E1 176.502} C_DIS
LIN {X 0.076,Y -475.458,Z 1339.777,A 0.000,B 0.000,C 90.000,E1 175.869} C_DIS
LIN {X 0.122,Y -474.567,Z 1339.774,A 0.000,B 0.000,C 90.000,E1 175.241} C_DIS
LIN {X 0.019,Y -473.031,Z 1339.769,A 0.000,B 0.000,C 90.000,E1 174.318} C_DIS
LIN {X 0.084,Y -471.832,Z 1339.765,A 0.000,B 0.000,C 90.000,E1 173.685} C_DIS
LIN {X 0.138,Y -470.312,Z 1339.762,A 0.000,B 0.000,C 90.000,E1 173.053} C_DIS
LIN {X -0.010,Y -467.322,Z 1339.756,A 0.000,B 0.000,C 90.000,E1 172.129} C_DIS
LIN {X -0.031,Y -465.655,Z 1339.754,A 0.000,B 0.000,C 90.000,E1 171.659} C_DIS
LIN {X -0.032,Y -462.798,Z 1339.750,A 0.000,B 0.000,C 90.000,E1 171.027} C_DIS
LIN {X 0.014,Y -459.658,Z 1339.747,A 0.000,B 0.000,C 90.000,E1 170.387} C_DIS
LIN {X -0.188,Y -454.034,Z 1339.741,A 0.000,B 0.000,C 90.000,E1 169.454} C_DIS
LIN {X -0.009,Y -447.963,Z 1339.736,A 0.000,B 0.000,C 90.000,E1 168.465} C_DIS
LIN {X -0.087,Y -439.393,Z 1339.729,A 0.000,B 0.000,C 90.000,E1 167.173} C_DIS
LIN {X -0.079,Y -428.549,Z 1339.719,A 0.000,B 0.000,C 90.000,E1 165.519} C_DIS
LIN {X 0.063,Y -420.103,Z 1339.712,A 0.000,B 0.000,C 90.000,E1 164.157} C_DIS
LIN {X -0.119,Y -416.792,Z 1339.708,A 0.000,B 0.000,C 90.000,E1 163.504} C_DIS
LIN {X -0.039,Y -416.257,Z 1339.707,A 0.000,B 0.000,C 90.000,E1 163.323} C_DIS
LIN {X -0.009,Y -414.823,Z 1339.704,A 0.000,B 0.000,C 90.000,E1 162.670} C_DIS
LIN {X -0.048,Y -414.821,Z 1339.704,A 0.000,B 0.000,C 90.000,E1 162.670} C_DIS
LIN {X 0.131,Y -415.447,Z 1339.702,A 0.000,B 0.000,C 90.000,E1 162.362} C_DIS
LIN {X 0.196,Y -417.308,Z 1339.701,A 0.000,B 0.000,C 90.000,E1 162.054} C_DIS
LIN {X -0.030,Y -417.748,Z 1339.700,A 0.000,B 0.000,C 90.000,E1 162.000} C_DIS
LIN {X -0.179,Y -423.264,Z 1339.697,A 0.000,B 0.000,C 90.000,E1 161.456} C_DIS
LIN {X 0.072,Y -431.868,Z 1339.693,A 0.000,B 0.000,C 90.000,E1 160.678} C_DIS
LIN {X -0.132,Y -447.385,Z 1339.686,A 0.000,B 0.000,C 90.000,E1 159.518} C_DIS
LIN {X 0.039,Y -458.250,Z 1339.682,A 0.000,B 0.000,C 90.000,E1 158.666} C_DIS
LIN {X -0.276,Y -466.063,Z 1339.678,A 0.000,B 0.000,C 90.000,E1 158.103} C_DIS
LIN {X 0.192,Y -476.716,Z 1339.673,A 0.000,B 0.000,C 90.000,E1 157.177} C_DIS
LIN {X 0.240,Y -482.633,Z 1339.671,A 0.000,B 0.000,C 90.000,E1 156.666} C_DIS
LIN {X -0.007,Y -488.396,Z 1339.668,A 0.000,B 0.000,C 90.000,E1 156.177} C_DIS
LIN {X 0.179,Y -495.444,Z 1339.664,A 0.000,B 0.000,C 90.000,E1 155.485} C_DIS
LIN {X 0.212,Y -502.322,Z 1339.660,A 0.000,B 0.000,C 90.000,E1 154.793} C_DIS
LIN {X -0.208,Y -508.760,Z 1339.656,A 0.000,B 0.000,C 90.000,E1 154.152} C_DIS
LIN {X 0.021,Y -513.749,Z 1339.653,A 0.000,B 0.000,C 90.000,E1 153.563} C_DIS
LIN {X -0.040,Y -517.450,Z 1339.651,A 0.000,B 0.000,C 90.000,E1 153.127} C_DIS
LIN {X -0.013,Y -521.946,Z 1339.647,A 0.000,B 0.000,C 90.000,E1 152.538} C_DIS
LIN {X -0.196,Y -526.047,Z 1339.644,A 0.000,B 0.000,C 90.000,E1 151.975} C_DIS
LIN {X -0.105,Y -529.642,Z 1339.641,A 0.000,B 0.000,C 90.000,E1 151.385} C_DIS
LIN {X -0.134,Y -533.205,Z 1339.637,A 0.000,B 0.000,C 90.000,E1 150.667} C_DIS
LIN {X 0.011,Y -535.601,Z 1339.634,A 0.000,B 0.000,C 90.000,E1 150.078} C_DIS
LIN {X -0.294,Y -537.648,Z 1339.631,A 0.000,B 0.000,C 90.000,E1 149.537} C_DIS
LIN {X -0.120,Y -540.260,Z 1339.626,A 0.000,B 0.000,C 90.000,E1 148.663} C_DIS
LIN {X 0.071,Y -541.857,Z 1339.623,A 0.000,B 0.000,C 90.000,E1 148.074} C_DIS
LIN {X -0.167,Y -543.889,Z 1339.618,A 0.000,B 0.000,C 90.000,E1 147.248} C_DIS
LIN {X 0.074,Y -545.570,Z 1339.613,A 0.000,B 0.000,C 90.000,E1 146.373} C_DIS
LIN {X 0.183,Y -547.026,Z 1339.609,A 0.000,B 0.000,C 90.000,E1 145.515} C_DIS
LIN {X 0.003,Y -548.140,Z 1339.604,A 0.000,B 0.000,C 90.000,E1 144.689} C_DIS
LIN {X 0.151,Y -549.082,Z 1339.599,A 0.000,B 0.000,C 90.000,E1 143.829} C_DIS
LIN {X 0.035,Y -550.019,Z 1339.593,A 0.000,B 0.000,C 90.000,E1 142.718} C_DIS
LIN {X -0.066,Y -551.073,Z 1339.584,A 0.000,B 0.000,C 90.000,E1 141.045} C_DIS
LIN {X 0.087,Y -551.799,Z 1339.577,A 0.000,B 0.000,C 90.000,E1 139.908} C_DIS
LIN {X 0.163,Y -554.260,Z 1339.560,A 0.000,B 0.000,C 90.000,E1 136.824} C_DIS
LIN {X 0.180,Y -554.935,Z 1339.558,A 0.000,B 0.000,C 90.000,E1 136.377} C_DIS
LIN {X 0.138,Y -554.959,Z 1339.558,A 0.000,B 0.000,C 90.000,E1 136.377} C_DIS
LIN {X -0.134,Y -555.933,Z 1339.557,A 0.000,B 0.000,C 90.000,E1 136.296} C_DIS
LIN {X 0.197,Y -557.270,Z 1339.556,A 0.000,B 0.000,C 90.000,E1 136.053} C_DIS
LIN {X -0.009,Y -557.540,Z 1339.556,A 0.000,B 0.000,C 90.000,E1 136.014} C_DIS
LIN {X 0.350,Y -557.584,Z 1339.556,A 0.000,B 0.000,C 90.000,E1 135.972} C_DIS
LIN {X 0.209,Y -559.268,Z 1339.555,A 0.000,B 0.000,C 90.000,E1 135.891} C_DIS
LIN {X 0.110,Y -561.963,Z 1339.555,A 0.000,B 0.000,C 90.000,E1 135.810} C_DIS
LIN {X 0.023,Y -569.752,Z 1339.553,A 0.000,B 0.000,C 90.000,E1 135.607} C_DIS
LIN {X 0.225,Y -572.876,Z 1339.553,A 0.000,B 0.000,C 90.000,E1 135.486} C_DIS
LIN {X -0.098,Y -575.781,Z 1339.552,A 0.000,B 0.000,C 90.000,E1 135.405} C_DIS
LIN {X 0.185,Y -578.546,Z 1339.552,A 0.000,B 0.000,C 90.000,E1 135.243} C_DIS
LIN {X 0.206,Y -581.522,Z 1339.551,A 0.000,B 0.000,C 90.000,E1 135.081} C_DIS
LIN {X 0.083,Y -584.495,Z 1339.550,A 0.000,B 0.000,C 90.000,E1 134.919} C_DIS
LIN {X -0.327,Y -588.836,Z 1339.548,A 0.000,B 0.000,C 90.000,E1 134.676} C_DIS
LIN {X -0.134,Y -593.122,Z 1339.546,A 0.000,B 0.000,C 90.000,E1 134.352} C_DIS
LIN {X -0.148,Y -597.377,Z 1339.545,A 0.000,B 0.000,C 90.000,E1 134.028} C_DIS
LIN {X -0.354,Y -601.357,Z 1339.543,A 0.000,B 0.000,C 90.000,E1 133.704} C_DIS
LIN {X 0.210,Y -606.390,Z 1339.540,A 0.000,B 0.000,C 90.000,E1 133.176} C_DIS
LIN {X 0.069,Y -611.325,Z 1339.537,A 0.000,B 0.000,C 90.000,E1 132.690} C_DIS
LIN {X 0.269,Y -614.900,Z 1339.535,A 0.000,B 0.000,C 90.000,E1 132.285} C_DIS
LIN {X 0.096,Y -620.221,Z 1339.532,A 0.000,B 0.000,C 90.000,E1 131.676} C_DIS
LIN {X -0.255,Y -625.524,Z 1339.528,A 0.000,B 0.000,C 90.000,E1 131.067} C_DIS
LIN {X -0.090,Y -630.599,Z 1339.525,A 0.000,B 0.000,C 90.000,E1 130.415} C_DIS
LIN {X 0.330,Y -639.899,Z 1339.518,A 0.000,B 0.000,C 90.000,E1 129.116} C_DIS
LIN {X 0.133,Y -645.077,Z 1339.513,A 0.000,B 0.000,C 90.000,E1 128.382} C_DIS
LIN {X -0.351,Y -649.280,Z 1339.510,A 0.000,B 0.000,C 90.000,E1 127.810} C_DIS
LIN {X 0.006,Y -652.529,Z 1339.507,A 0.000,B 0.000,C 90.000,E1 127.282} C_DIS
LIN {X 0.058,Y -657.286,Z 1339.503,A 0.000,B 0.000,C 90.000,E1 126.537} C_DIS
LIN {X 0.024,Y -661.680,Z 1339.499,A 0.000,B 0.000,C 90.000,E1 125.804} C_DIS
LIN {X 0.072,Y -664.433,Z 1339.496,A 0.000,B 0.000,C 90.000,E1 125.311} C_DIS
LIN {X 0.195,Y -667.470,Z 1339.493,A 0.000,B 0.000,C 90.000,E1 124.692} C_DIS
LIN {X 0.280,Y -669.742,Z 1339.490,A 0.000,B 0.000,C 90.000,E1 124.199} C_DIS
LIN {X -0.038,Y -672.830,Z 1339.486,A 0.000,B 0.000,C 90.000,E1 123.499} C_DIS
LIN {X 0.233,Y -675.376,Z 1339.482,A 0.000,B 0.000,C 90.000,E1 122.752} C_DIS
LIN {X -0.042,Y -677.599,Z 1339.478,A 0.000,B 0.000,C 90.000,E1 122.054} C_DIS
LIN {X 0.108,Y -680.170,Z 1339.473,A 0.000,B 0.000,C 90.000,E1 121.082} C_DIS
LIN {X -0.135,Y -681.794,Z 1339.469,A 0.000,B 0.000,C 90.000,E1 120.384} C_DIS
LIN {X -0.123,Y -683.069,Z 1339.465,A 0.000,B 0.000,C 90.000,E1 119.667} C_DIS
LIN {X -0.095,Y -684.006,Z 1339.461,A 0.000,B 0.000,C 90.000,E1 118.949} C_DIS
LIN {X 0.158,Y -684.631,Z 1339.456,A 0.000,B 0.000,C 90.000,E1 117.975} C_DIS
LIN {X 0.202,Y -684.797,Z 1339.452,A 0.000,B 0.000,C 90.000,E1 117.257} C_DIS
LIN {X 0.154,Y -684.672,Z 1339.446,A 0.000,B 0.000,C 90.000,E1 116.309} C_DIS
LIN {X -0.026,Y -684.483,Z 1339.444,A 0.000,B 0.000,C 90.000,E1 115.848} C_DIS
LIN {X 0.406,Y -684.128,Z 1339.441,A 0.000,B 0.000,C 90.000,E1 115.335} C_DIS
LIN {X -0.075,Y -683.574,Z 1339.438,A 0.000,B 0.000,C 90.000,E1 114.899} C_DIS
LIN {X 0.348,Y -682.608,Z 1339.436,A 0.000,B 0.000,C 90.000,E1 114.387} C_DIS
LIN {X -0.346,Y -682.050,Z 1339.434,A 0.000,B 0.000,C 90.000,E1 114.207} C_DIS
LIN {X -0.109,Y -679.615,Z 1339.431,A 0.000,B 0.000,C 90.000,E1 113.590} C_DIS
LIN {X -0.008,Y -678.794,Z 1339.430,A 0.000,B 0.000,C 90.000,E1 113.462} C_DIS
LIN {X 0.372,Y -674.675,Z 1339.428,A 0.000,B 0.000,C 90.000,E1 112.950} C_DIS
LIN {X -0.422,Y -673.193,Z 1339.427,A 0.000,B 0.000,C 90.000,E1 112.898} C_DIS
LIN {X -0.227,Y -667.709,Z 1339.425,A 0.000,B 0.000,C 90.000,E1 112.589} C_DIS
LIN {X 0.098,Y -664.539,Z 1339.425,A 0.000,B 0.000,C 90.000,E1 112.408} C_DIS
LIN {X -0.137,Y -659.982,Z 1339.424,A 0.000,B 0.000,C 90.000,E1 112.280} C_DIS
LIN {X 0.077,Y -657.663,Z 1339.423,A 0.000,B 0.000,C 90.000,E1 112.206} C_DIS
LIN {X 0.056,Y -644.060,Z 1339.422,A 0.000,B 0.000,C 90.000,E1 111.972} C_DIS
LIN {X -0.061,Y -640.040,Z 1339.422,A 0.000,B 0.000,C 90.000,E1 111.897} C_DIS
LIN {X -0.114,Y -639.908,Z 1339.422,A 0.000,B 0.000,C 90.000,E1 111.897} C_DIS
LIN {X 0.142,Y -642.991,Z 1339.419,A 0.000,B 0.000,C 90.000,E1 111.461} C_DIS
LIN {X 0.049,Y -647.087,Z 1339.417,A 0.000,B 0.000,C 90.000,E1 110.972} C_DIS
LIN {X -0.017,Y -650.934,Z 1339.414,A 0.000,B 0.000,C 90.000,E1 110.482} C_DIS
LIN {X -0.039,Y -655.014,Z 1339.410,A 0.000,B 0.000,C 90.000,E1 109.866} C_DIS
LIN {X -0.297,Y -657.874,Z 1339.408,A 0.000,B 0.000,C 90.000,E1 109.396} C_DIS
LIN {X -0.216,Y -661.453,Z 1339.404,A 0.000,B 0.000,C 90.000,E1 108.652} C_DIS
LIN {X 0.310,Y -664.589,Z 1339.400,A 0.000,B 0.000,C 90.000,E1 107.873} C_DIS
LIN {X 0.040,Y -667.420,Z 1339.395,A 0.000,B 0.000,C 90.000,E1 107.166} C_DIS
LIN {X -0.003,Y -669.947,Z 1339.391,A 0.000,B 0.000,C 90.000,E1 106.441} C_DIS
LIN {X -0.144,Y -671.461,Z 1339.389,A 0.000,B 0.000,C 90.000,E1 105.969} C_DIS
LIN {X -0.158,Y -673.354,Z 1339.385,A 0.000,B 0.000,C 90.000,E1 105.245} C_DIS
LIN {X -0.333,Y -674.949,Z 1339.381,A 0.000,B 0.000,C 90.000,E1 104.537} C_DIS
LIN {X 0.215,Y -675.782,Z 1339.378,A 0.000,B 0.000,C 90.000,E1 104.008} C_DIS
LIN {X 0.116,Y -676.445,Z 1339.375,A 0.000,B 0.000,C 90.000,E1 103.536} C_DIS
LIN {X 0.020,Y -676.928,Z 1339.373,A 0.000,B 0.000,C 90.000,E1 103.063} C_DIS
LIN {X -0.122,Y -677.167,Z 1339.369,A 0.000,B 0.000,C 90.000,E1 102.355} C_DIS
LIN {X -0.218,Y -677.177,Z 1339.366,A 0.000,B 0.000,C 90.000,E1 101.883} C_DIS
LIN {X 0.213,Y -677.004,Z 1339.363,A 0.000,B 0.000,C 90.000,E1 101.366} C_DIS
LIN {X 0.115,Y -676.588,Z 1339.361,A 0.000,B 0.000,C 90.000,E1 100.894} C_DIS
LIN {X -0.114,Y -675.964,Z 1339.358,A 0.000,B 0.000,C 90.000,E1 100.433} C_DIS
LIN {X -0.281,Y -674.539,Z 1339.354,A 0.000,B 0.000,C 90.000,E1 99.726} C_DIS
LIN {X 0.148,Y -673.337,Z 1339.351,A 0.000,B 0.000,C 90.000,E1 99.208} C_DIS
LIN {X -0.090,Y -671.774,Z 1339.349,A 0.000,B 0.000,C 90.000,E1 98.746} C_DIS
LIN {X -0.238,Y -669.894,Z 1339.346,A 0.000,B 0.000,C 90.000,E1 98.276} C_DIS
LIN {X -0.012,Y -666.713,Z 1339.342,A 0.000,B 0.000,C 90.000,E1 97.530} C_DIS
LIN {X -0.295,Y -663.794,Z 1339.339,A 0.000,B 0.000,C 90.000,E1 96.947} C_DIS
LIN {X -0.125,Y -659.972,Z 1339.334,A 0.000,B 0.000,C 90.000,E1 96.201} C_DIS
LIN {X 0.011,Y -655.626,Z 1339.330,A 0.000,B 0.000,C 90.000,E1 95.454} C_DIS
LIN {X -0.336,Y -652.538,Z 1339.328,A 0.000,B 0.000,C 90.000,E1 94.992} C_DIS
LIN {X -0.163,Y -648.273,Z 1339.324,A 0.000,B 0.000,C 90.000,E1 94.359} C_DIS
LIN {X 0.085,Y -644.652,Z 1339.321,A 0.000,B 0.000,C 90.000,E1 93.841} C_DIS
LIN {X 0.265,Y -640.745,Z 1339.319,A 0.000,B 0.000,C 90.000,E1 93.326} C_DIS
LIN {X -0.183,Y -636.283,Z 1339.316,A 0.000,B 0.000,C 90.000,E1 92.865} C_DIS
LIN {X -0.084,Y -630.099,Z 1339.312,A 0.000,B 0.000,C 90.000,E1 92.236} C_DIS
LIN {X -0.193,Y -618.778,Z 1339.306,A 0.000,B 0.000,C 90.000,E1 91.146} C_DIS
LIN {X 0.186,Y -614.576,Z 1339.304,A 0.000,B 0.000,C 90.000,E1 90.745} C_DIS
LIN {X 0.153,Y -608.991,Z 1339.302,A 0.000,B 0.000,C 90.000,E1 90.286} C_DIS
LIN {X 0.119,Y -602.553,Z 1339.299,A 0.000,B 0.000,C 90.000,E1 89.885} C_DIS
LIN {X 0.098,Y -595.656,Z 1339.298,A 0.000,B 0.000,C 90.000,E1 89.542} C_DIS
LIN {X -0.191,Y -586.851,Z 1339.296,A 0.000,B 0.000,C 90.000,E1 89.198} C_DIS
LIN {X 0.170,Y -583.386,Z 1339.295,A 0.000,B 0.000,C 90.000,E1 89.026} C_DIS
LIN {X -0.200,Y -577.530,Z 1339.293,A 0.000,B 0.000,C 90.000,E1 88.797} C_DIS
LIN {X 0.068,Y -573.458,Z 1339.292,A 0.000,B 0.000,C 90.000,E1 88.453} C_DIS
LIN {X -0.252,Y -573.195,Z 1339.291,A 0.000,B 0.000,C 90.000,E1 88.453} C_DIS
LIN {X -0.288,Y -573.185,Z 1339.291,A 0.000,B 0.000,C 90.000,E1 88.453} C_DIS
LIN {X -0.140,Y -572.648,Z 1339.290,A 0.000,B 0.000,C 90.000,E1 88.224} C_DIS
LIN {X 0.235,Y -572.486,Z 1339.289,A 0.000,B 0.000,C 90.000,E1 88.051} C_DIS
LIN {X -0.057,Y -572.526,Z 1339.287,A 0.000,B 0.000,C 90.000,E1 87.650} C_DIS
LIN {X 0.149,Y -574.789,Z 1339.273,A 0.000,B 0.000,C 90.000,E1 85.179} C_DIS
LIN {X -0.097,Y -577.548,Z 1339.260,A 0.000,B 0.000,C 90.000,E1 82.761} C_DIS
LIN {X 0.230,Y -579.185,Z 1339.252,A 0.000,B 0.000,C 90.000,E1 81.376} C_DIS
LIN {X 0.099,Y -580.847,Z 1339.245,A 0.000,B 0.000,C 90.000,E1 80.038} C_DIS
LIN {X 0.228,Y -582.568,Z 1339.236,A 0.000,B 0.000,C 90.000,E1 78.409} C_DIS
LIN {X -0.305,Y -583.818,Z 1339.228,A 0.000,B 0.000,C 90.000,E1 77.117} C_DIS
LIN {X -0.109,Y -584.955,Z 1339.221,A 0.000,B 0.000,C 90.000,E1 75.755} C_DIS
LIN {X 0.112,Y -585.900,Z 1339.213,A 0.000,B 0.000,C 90.000,E1 74.393} C_DIS
LIN {X -0.223,Y -586.837,Z 1339.206,A 0.000,B 0.000,C 90.000,E1 73.087} C_DIS
LIN {X 0.039,Y -587.815,Z 1339.197,A 0.000,B 0.000,C 90.000,E1 71.456} C_DIS
LIN {X 0.097,Y -588.648,Z 1339.190,A 0.000,B 0.000,C 90.000,E1 70.115} C_DIS
LIN {X -0.279,Y -589.832,Z 1339.179,A 0.000,B 0.000,C 90.000,E1 68.284} C_DIS
LIN {X 0.245,Y -591.256,Z 1339.167,A 0.000,B 0.000,C 90.000,E1 66.102} C_DIS
LIN {X -0.073,Y -592.431,Z 1339.159,A 0.000,B 0.000,C 90.000,E1 64.537} C_DIS
LIN {X -0.030,Y -593.395,Z 1339.151,A 0.000,B 0.000,C 90.000,E1 63.204} C_DIS
LIN {X 0.207,Y -595.309,Z 1339.138,A 0.000,B 0.000,C 90.000,E1 60.795} C_DIS
LIN {X 0.042,Y -596.579,Z 1339.131,A 0.000,B 0.000,C 90.000,E1 59.488} C_DIS
LIN {X -0.089,Y -598.187,Z 1339.122,A 0.000,B 0.000,C 90.000,E1 57.916} C_DIS
LIN {X -0.171,Y -599.780,Z 1339.113,A 0.000,B 0.000,C 90.000,E1 56.342} C_DIS
LIN {X -0.230,Y -601.401,Z 1339.104,A 0.000,B 0.000,C 90.000,E1 54.769} C_DIS
LIN {X -0.073,Y -602.380,Z 1339.098,A 0.000,B 0.000,C 90.000,E1 53.703} C_DIS
LIN {X -0.126,Y -603.584,Z 1339.091,A 0.000,B 0.000,C 90.000,E1 52.396} C_DIS
LIN {X 0.104,Y -604.693,Z 1339.082,A 0.000,B 0.000,C 90.000,E1 50.803} C_DIS
LIN {X 0.008,Y -605.524,Z 1339.075,A 0.000,B 0.000,C 90.000,E1 49.504} C_DIS
LIN {X 0.388,Y -606.019,Z 1339.068,A 0.000,B 0.000,C 90.000,E1 48.162} C_DIS
